gfCNCPoint5[22802] = {X 520.5269, Y 35.5815, Z -7.1667, A 0.000, B 0.000, C 0.000 }
gfCNCPoint5[22803] = {X 521.3531, Y 35.6727, Z -7.1667, A 0.000, B 0.000, C 0.000 }
gfCNCPoint5[22804] = {X 522.1466, Y 35.9205, Z -7.1667, A 0.000, B 0.000, C 0.000 }
gfCNCPoint5[22805] = {X 522.8780, Y 36.3157, Z -7.1667, A 0.000, B 0.000, C 0.000 }
gfCNCPoint5[22806] = {X 523.5201, Y 36.8436, Z -7.1667, A 0.000, B 0.000, C 0.000 }
gfCNCPoint5[22807] = {X 524.0492, Y 37.4848, Z -7.1667, A 0.000, B 0.000, C 0.000 }
gfCNCPoint5[22808] = {X 534.6319, Y 37.4851, Z -7.1667, A 0.000, B 0.000, C 0.000 }
gfCNCPoint5[22809] = {X 534.6319, Y 33.9662, Z -7.1667, A 0.000, B 0.000, C 0.000 }
gfCNCPoint5[22810] = {X 530.1083, Y 33.9675, Z -7.1667, A 0.000, B 0.000, C 0.000 }
gfCNCPoint5[22811] = {X 529.5761, Y 34.6112, Z -7.1667, A 0.000, B 0.000, C 0.000 }
gfCNCPoint5[22812] = {X 528.9300, Y 35.1404, Z -7.1667, A 0.000, B 0.000, C 0.000 }
gfCNCPoint5[22813] = {X 528.1941, Y 35.5354, Z -7.1667, A 0.000, B 0.000, C 0.000 }
gfCNCPoint5[22814] = {X 527.3960, Y 35.7814, Z -7.1667, A 0.000, B 0.000, C 0.000 }
gfCNCPoint5[22815] = {X 526.5655, Y 35.8693, Z -7.1667, A 0.000, B 0.000, C 0.000 }
gfCNCPoint5[22816] = {X 525.8868, Y 35.8694, Z -7.1667, A 0.000, B 0.000, C 0.000 }
gfCNCPoint5[22817] = {X 524.9255, Y 35.7611, Z -7.1667, A 0.000, B 0.000, C 0.000 }
gfCNCPoint5[22818] = {X 524.0124, Y 35.4416, Z -7.1667, A 0.000, B 0.000, C 0.000 }
gfCNCPoint5[22819] = {X 523.1933, Y 34.9270, Z -7.1667, A 0.000, B 0.000, C 0.000 }
gfCNCPoint5[22820] = {X 522.5092, Y 34.2429, Z -7.1667, A 0.000, B 0.000, C 0.000 }
gfCNCPoint5[22821] = {X 521.9946, Y 33.4238, Z -7.1667, A 0.000, B 0.000, C 0.000 }
gfCNCPoint5[22822] = {X 521.6751, Y 32.5107, Z -7.1667, A 0.000, B 0.000, C 0.000 }
gfCNCPoint5[22823] = {X 521.5668, Y 31.5495, Z -7.1667, A 0.000, B 0.000, C 0.000 }
gfCNCPoint5[22824] = {X 521.5668, Y 24.5714, Z -7.1667, A 0.000, B 0.000, C 0.000 }
gfCNCPoint5[22825] = {X 521.6739, Y 23.6153, Z -7.1667, A 0.000, B 0.000, C 0.000 }
gfCNCPoint5[22826] = {X 521.9900, Y 22.7066, Z -7.1667, A 0.000, B 0.000, C 0.000 }
gfCNCPoint5[22827] = {X 522.4994, Y 21.8904, Z -7.1667, A 0.000, B 0.000, C 0.000 }
gfCNCPoint5[22828] = {X 523.1768, Y 21.2071, Z -7.1667, A 0.000, B 0.000, C 0.000 }
gfCNCPoint5[22829] = {X 523.9886, Y 20.6908, Z -7.1667, A 0.000, B 0.000, C 0.000 }
gfCNCPoint5[22830] = {X 524.8946, Y 20.3669, Z -7.1667, A 0.000, B 0.000, C 0.000 }
gfCNCPoint5[22831] = {X 525.8498, Y 20.2516, Z -7.1667, A 0.000, B 0.000, C 0.000 }
gfCNCPoint5[22832] = {X 526.5695, Y 20.2516, Z -7.1667, A 0.000, B 0.000, C 0.000 }
gfCNCPoint5[22833] = {X 527.3943, Y 20.3391, Z -7.1667, A 0.000, B 0.000, C 0.000 }
gfCNCPoint5[22834] = {X 528.1872, Y 20.5826, Z -7.1667, A 0.000, B 0.000, C 0.000 }
gfCNCPoint5[22835] = {X 528.9190, Y 20.9731, Z -7.1667, A 0.000, B 0.000, C 0.000 }
gfCNCPoint5[22836] = {X 529.5626, Y 21.4964, Z -7.1667, A 0.000, B 0.000, C 0.000 }
gfCNCPoint5[22837] = {X 530.0944, Y 22.1329, Z -7.1667, A 0.000, B 0.000, C 0.000 }
gfCNCPoint5[22838] = {X 534.6319, Y 22.1331, Z -7.1667, A 0.000, B 0.000, C 0.000 }
gfCNCPoint5[22839] = {X 534.6319, Y 19.7026, Z -7.1667, A 0.000, B 0.000, C 0.000 }
gfCNCPoint5[22840] = {X 524.1915, Y 19.7025, Z -7.1667, A 0.000, B 0.000, C 0.000 }
gfCNCPoint5[22841] = {X 523.6591, Y 20.3468, Z -7.1667, A 0.000, B 0.000, C 0.000 }
gfCNCPoint5[22842] = {X 523.0125, Y 20.8765, Z -7.1667, A 0.000, B 0.000, C 0.000 }
gfCNCPoint5[22843] = {X 522.2760, Y 21.2718, Z -7.1667, A 0.000, B 0.000, C 0.000 }
gfCNCPoint5[22844] = {X 521.4772, Y 21.5179, Z -7.1667, A 0.000, B 0.000, C 0.000 }
gfCNCPoint5[22845] = {X 520.6460, Y 21.6056, Z -7.1667, A 0.000, B 0.000, C 0.000 }
gfCNCPoint5[22846] = {X 519.9691, Y 21.6057, Z -7.1667, A 0.000, B 0.000, C 0.000 }
gfCNCPoint5[22847] = {X 519.0078, Y 21.4974, Z -7.1667, A 0.000, B 0.000, C 0.000 }
gfCNCPoint5[22848] = {X 518.0947, Y 21.1779, Z -7.1667, A 0.000, B 0.000, C 0.000 }
gfCNCPoint5[22849] = {X 517.2756, Y 20.6632, Z -7.1667, A 0.000, B 0.000, C 0.000 }
gfCNCPoint5[22850] = {X 516.5916, Y 19.9792, Z -7.1667, A 0.000, B 0.000, C 0.000 }
gfCNCPoint5[22851] = {X 516.0769, Y 19.1601, Z -7.1667, A 0.000, B 0.000, C 0.000 }
gfCNCPoint5[22852] = {X 515.7574, Y 18.2470, Z -7.1667, A 0.000, B 0.000, C 0.000 }
gfCNCPoint5[22853] = {X 515.6491, Y 17.2857, Z -7.1667, A 0.000, B 0.000, C 0.000 }
gfCNCPoint5[22854] = {X 515.6491, Y 10.3077, Z -7.1667, A 0.000, B 0.000, C 0.000 }
gfCNCPoint5[22855] = {X 515.7562, Y 9.3519, Z -7.1667, A 0.000, B 0.000, C 0.000 }
gfCNCPoint5[22856] = {X 516.0720, Y 8.4435, Z -7.1667, A 0.000, B 0.000, C 0.000 }
gfCNCPoint5[22857] = {X 516.5811, Y 7.6275, Z -7.1667, A 0.000, B 0.000, C 0.000 }
gfCNCPoint5[22858] = {X 517.2580, Y 6.9443, Z -7.1667, A 0.000, B 0.000, C 0.000 }
gfCNCPoint5[22859] = {X 518.0693, Y 6.4278, Z -7.1667, A 0.000, B 0.000, C 0.000 }
gfCNCPoint5[22860] = {X 518.9748, Y 6.1037, Z -7.1667, A 0.000, B 0.000, C 0.000 }
gfCNCPoint5[22861] = {X 519.9296, Y 5.9879, Z -7.1667, A 0.000, B 0.000, C 0.000 }
gfCNCPoint5[22862] = {X 520.6502, Y 5.9879, Z -7.1667, A 0.000, B 0.000, C 0.000 }
gfCNCPoint5[22863] = {X 521.4754, Y 6.0751, Z -7.1667, A 0.000, B 0.000, C 0.000 }
gfCNCPoint5[22864] = {X 522.2687, Y 6.3185, Z -7.1667, A 0.000, B 0.000, C 0.000 }
gfCNCPoint5[22865] = {X 523.0008, Y 6.7091, Z -7.1667, A 0.000, B 0.000, C 0.000 }
gfCNCPoint5[22866] = {X 523.6448, Y 7.2324, Z -7.1667, A 0.000, B 0.000, C 0.000 }
gfCNCPoint5[22867] = {X 524.1768, Y 7.8692, Z -7.1667, A 0.000, B 0.000, C 0.000 }
gfCNCPoint5[22868] = {X 533.9633, Y 7.8694, Z -7.1667, A 0.000, B 0.000, C 0.000 }
gfCNCPoint5[22869] = {X 533.9634, Y 3.8694, Z -7.1667, A 0.000, B 0.000, C 0.000 }
gfCNCPoint5[22870] = {X 533.9633, Y 7.9494, Z -7.1667, A 0.000, B 0.000, C 0.000 }
gfCNCPoint5[22871] = {X 543.7510, Y 7.9496, Z -7.1667, A 0.000, B 0.000, C 0.000 }
gfCNCPoint5[22872] = {X 544.7134, Y 8.0333, Z -7.1667, A 0.000, B 0.000, C 0.000 }
gfCNCPoint5[22873] = {X 545.6320, Y 8.3325, Z -7.1667, A 0.000, B 0.000, C 0.000 }
gfCNCPoint5[22874] = {X 546.4591, Y 8.8316, Z -7.1667, A 0.000, B 0.000, C 0.000 }
gfCNCPoint5[22875] = {X 547.1520, Y 9.5048, Z -7.1667, A 0.000, B 0.000, C 0.000 }
gfCNCPoint5[22876] = {X 547.6747, Y 10.3173, Z -7.1667, A 0.000, B 0.000, C 0.000 }
gfCNCPoint5[22877] = {X 548.0001, Y 11.2269, Z -7.1667, A 0.000, B 0.000, C 0.000 }
gfCNCPoint5[22878] = {X 548.1114, Y 12.1865, Z -7.1667, A 0.000, B 0.000, C 0.000 }
gfCNCPoint5[22879] = {X 548.1112, Y 13.0217, Z -7.1667, A 0.000, B 0.000, C 0.000 }
gfCNCPoint5[22880] = {X 548.0029, Y 13.9312, Z -7.1667, A 0.000, B 0.000, C 0.000 }
gfCNCPoint5[22881] = {X 547.7018, Y 14.7962, Z -7.1667, A 0.000, B 0.000, C 0.000 }
gfCNCPoint5[22882] = {X 547.2220, Y 15.5764, Z -7.1667, A 0.000, B 0.000, C 0.000 }
gfCNCPoint5[22883] = {X 546.5858, Y 16.2353, Z -7.1667, A 0.000, B 0.000, C 0.000 }
gfCNCPoint5[22884] = {X 546.5850, Y 40.9520, Z -7.1667, A 0.000, B 0.000, C 0.000 }
gfCNCPoint5[22885] = {X 546.6353, Y 40.9934, Z -7.1667, A 0.000, B 0.000, C 0.000 }
gfCNCPoint5[22886] = {X 547.2529, Y 41.6508, Z -7.1667, A 0.000, B 0.000, C 0.000 }
gfCNCPoint5[22887] = {X 547.7175, Y 42.4239, Z -7.1667, A 0.000, B 0.000, C 0.000 }
gfCNCPoint5[22888] = {X 548.0080, Y 43.2779, Z -7.1667, A 0.000, B 0.000, C 0.000 }
gfCNCPoint5[22889] = {X 548.1113, Y 44.1740, Z -7.1667, A 0.000, B 0.000, C 0.000 }
gfCNCPoint5[22890] = {X 548.1114, Y 45.0003, Z -7.1667, A 0.000, B 0.000, C 0.000 }
gfCNCPoint5[22891] = {X 548.0001, Y 45.9599, Z -7.1667, A 0.000, B 0.000, C 0.000 }
gfCNCPoint5[22892] = {X 547.6746, Y 46.8695, Z -7.1667, A 0.000, B 0.000, C 0.000 }
gfCNCPoint5[22893] = {X 547.1519, Y 47.6819, Z -7.1667, A 0.000, B 0.000, C 0.000 }
gfCNCPoint5[22894] = {X 546.4591, Y 48.3551, Z -7.1667, A 0.000, B 0.000, C 0.000 }
gfCNCPoint5[22895] = {X 545.6320, Y 48.8541, Z -7.1667, A 0.000, B 0.000, C 0.000 }
gfCNCPoint5[22896] = {X 544.7134, Y 49.1533, Z -7.1667, A 0.000, B 0.000, C 0.000 }
gfCNCPoint5[22897] = {X 543.7510, Y 49.2369, Z -7.1667, A 0.000, B 0.000, C 0.000 }
gfCNCPoint5[22898] = {X 524.0041, Y 49.2373, Z -7.1667, A 0.000, B 0.000, C 0.000 }
gfCNCPoint5[22899] = {X 523.4672, Y 49.8705, Z -7.1667, A 0.000, B 0.000, C 0.000 }
gfCNCPoint5[22900] = {X 522.8209, Y 50.3914, Z -7.1667, A 0.000, B 0.000, C 0.000 }
gfCNCPoint5[22901] = {X 522.0882, Y 50.7816, Z -7.1667, A 0.000, B 0.000, C 0.000 }
gfCNCPoint5[22902] = {X 521.2952, Y 51.0271, Z -7.1667, A 0.000, B 0.000, C 0.000 }
gfCNCPoint5[22903] = {X 520.4702, Y 51.1191, Z -7.1667, A 0.000, B 0.000, C 0.000 }
gfCNCPoint5[22904] = {X 519.7998, Y 51.1191, Z -7.1667, A 0.000, B 0.000, C 0.000 }
gfCNCPoint5[22905] = {X 518.8563, Y 51.0128, Z -7.1667, A 0.000, B 0.000, C 0.000 }
gfCNCPoint5[22906] = {X 517.9601, Y 50.6992, Z -7.1667, A 0.000, B 0.000, C 0.000 }
gfCNCPoint5[22907] = {X 517.1562, Y 50.1941, Z -7.1667, A 0.000, B 0.000, C 0.000 }
gfCNCPoint5[22908] = {X 516.4848, Y 49.5227, Z -7.1667, A 0.000, B 0.000, C 0.000 }
gfCNCPoint5[22909] = {X 515.9797, Y 48.7188, Z -7.1667, A 0.000, B 0.000, C 0.000 }
gfCNCPoint5[22910] = {X 515.6661, Y 47.8226, Z -7.1667, A 0.000, B 0.000, C 0.000 }
gfCNCPoint5[22911] = {X 515.5598, Y 46.8791, Z -7.1667, A 0.000, B 0.000, C 0.000 }
gfCNCPoint5[22912] = {X 515.5598, Y 39.9011, Z -7.1667, A 0.000, B 0.000, C 0.000 }
gfCNCPoint5[22913] = {X 515.6649, Y 38.9628, Z -7.1667, A 0.000, B 0.000, C 0.000 }
gfCNCPoint5[22914] = {X 515.9751, Y 38.0710, Z -7.1667, A 0.000, B 0.000, C 0.000 }
gfCNCPoint5[22915] = {X 516.4749, Y 37.2700, Z -7.1667, A 0.000, B 0.000, C 0.000 }
gfCNCPoint5[22916] = {X 517.1395, Y 36.5995, Z -7.1667, A 0.000, B 0.000, C 0.000 }
gfCNCPoint5[22917] = {X 517.9361, Y 36.0926, Z -7.1667, A 0.000, B 0.000, C 0.000 }
gfCNCPoint5[22918] = {X 518.8251, Y 35.7746, Z -7.1667, A 0.000, B 0.000, C 0.000 }
gfCNCPoint5[22919] = {X 519.7624, Y 35.6613, Z -7.1667, A 0.000, B 0.000, C 0.000 }
gfCNCPoint5[22920] = {X 520.5258, Y 35.6615, Z -7.1667, A 0.000, B 0.000, C 0.000 }
gfCNCPoint5[22921] = {X 521.3450, Y 35.7528, Z -7.1667, A 0.000, B 0.000, C 0.000 }
gfCNCPoint5[22922] = {X 522.1312, Y 36.0008, Z -7.1667, A 0.000, B 0.000, C 0.000 }
gfCNCPoint5[22923] = {X 522.8544, Y 36.3963, Z -7.1667, A 0.000, B 0.000, C 0.000 }
gfCNCPoint5[22924] = {X 523.4875, Y 36.9243, Z -7.1667, A 0.000, B 0.000, C 0.000 }
gfCNCPoint5[22925] = {X 524.0064, Y 37.5648, Z -7.1667, A 0.000, B 0.000, C 0.000 }
gfCNCPoint5[22926] = {X 534.7119, Y 37.5651, Z -7.1667, A 0.000, B 0.000, C 0.000 }
gfCNCPoint5[22927] = {X 534.7119, Y 33.8862, Z -7.1667, A 0.000, B 0.000, C 0.000 }
gfCNCPoint5[22928] = {X 530.0654, Y 33.8860, Z -7.1667, A 0.000, B 0.000, C 0.000 }
gfCNCPoint5[22929] = {X 530.0414, Y 33.9236, Z -7.1667, A 0.000, B 0.000, C 0.000 }
gfCNCPoint5[22930] = {X 529.5191, Y 34.5550, Z -7.1667, A 0.000, B 0.000, C 0.000 }
gfCNCPoint5[22931] = {X 528.8850, Y 35.0742, Z -7.1667, A 0.000, B 0.000, C 0.000 }
gfCNCPoint5[22932] = {X 528.1629, Y 35.4617, Z -7.1667, A 0.000, B 0.000, C 0.000 }
gfCNCPoint5[22933] = {X 527.3797, Y 35.7031, Z -7.1667, A 0.000, B 0.000, C 0.000 }
gfCNCPoint5[22934] = {X 526.5648, Y 35.7893, Z -7.1667, A 0.000, B 0.000, C 0.000 }
gfCNCPoint5[22935] = {X 525.8868, Y 35.7894, Z -7.1667, A 0.000, B 0.000, C 0.000 }
gfCNCPoint5[22936] = {X 524.9433, Y 35.6831, Z -7.1667, A 0.000, B 0.000, C 0.000 }
gfCNCPoint5[22937] = {X 524.0471, Y 35.3696, Z -7.1667, A 0.000, B 0.000, C 0.000 }
gfCNCPoint5[22938] = {X 523.2432, Y 34.8644, Z -7.1667, A 0.000, B 0.000, C 0.000 }
gfCNCPoint5[22939] = {X 522.5718, Y 34.1930, Z -7.1667, A 0.000, B 0.000, C 0.000 }
gfCNCPoint5[22940] = {X 522.0666, Y 33.3891, Z -7.1667, A 0.000, B 0.000, C 0.000 }
gfCNCPoint5[22941] = {X 521.7531, Y 32.4929, Z -7.1667, A 0.000, B 0.000, C 0.000 }
gfCNCPoint5[22942] = {X 521.6468, Y 31.5495, Z -7.1667, A 0.000, B 0.000, C 0.000 }
gfCNCPoint5[22943] = {X 521.6468, Y 24.5714, Z -7.1667, A 0.000, B 0.000, C 0.000 }
gfCNCPoint5[22944] = {X 521.7519, Y 23.6330, Z -7.1667, A 0.000, B 0.000, C 0.000 }
gfCNCPoint5[22945] = {X 522.0622, Y 22.7411, Z -7.1667, A 0.000, B 0.000, C 0.000 }
gfCNCPoint5[22946] = {X 522.5621, Y 21.9400, Z -7.1667, A 0.000, B 0.000, C 0.000 }
gfCNCPoint5[22947] = {X 523.2270, Y 21.2694, Z -7.1667, A 0.000, B 0.000, C 0.000 }
gfCNCPoint5[22948] = {X 524.0238, Y 20.7626, Z -7.1667, A 0.000, B 0.000, C 0.000 }
gfCNCPoint5[22949] = {X 524.9130, Y 20.4448, Z -7.1667, A 0.000, B 0.000, C 0.000 }
gfCNCPoint5[22950] = {X 525.8505, Y 20.3316, Z -7.1667, A 0.000, B 0.000, C 0.000 }
gfCNCPoint5[22951] = {X 526.5687, Y 20.3316, Z -7.1667, A 0.000, B 0.000, C 0.000 }
gfCNCPoint5[22952] = {X 527.3865, Y 20.4192, Z -7.1667, A 0.000, B 0.000, C 0.000 }
gfCNCPoint5[22953] = {X 528.1720, Y 20.6630, Z -7.1667, A 0.000, B 0.000, C 0.000 }
gfCNCPoint5[22954] = {X 528.8957, Y 21.0538, Z -7.1667, A 0.000, B 0.000, C 0.000 }
gfCNCPoint5[22955] = {X 529.5303, Y 21.5770, Z -7.1667, A 0.000, B 0.000, C 0.000 }
gfCNCPoint5[22956] = {X 530.0519, Y 22.2129, Z -7.1667, A 0.000, B 0.000, C 0.000 }
gfCNCPoint5[22957] = {X 534.7119, Y 22.2131, Z -7.1667, A 0.000, B 0.000, C 0.000 }
gfCNCPoint5[22958] = {X 534.7119, Y 19.6226, Z -7.1667, A 0.000, B 0.000, C 0.000 }
gfCNCPoint5[22959] = {X 524.1486, Y 19.6225, Z -7.1667, A 0.000, B 0.000, C 0.000 }
gfCNCPoint5[22960] = {X 524.1252, Y 19.6577, Z -7.1667, A 0.000, B 0.000, C 0.000 }
gfCNCPoint5[22961] = {X 523.6026, Y 20.2901, Z -7.1667, A 0.000, B 0.000, C 0.000 }
gfCNCPoint5[22962] = {X 522.9680, Y 20.8100, Z -7.1667, A 0.000, B 0.000, C 0.000 }
gfCNCPoint5[22963] = {X 522.2452, Y 21.1980, Z -7.1667, A 0.000, B 0.000, C 0.000 }
gfCNCPoint5[22964] = {X 521.4612, Y 21.4396, Z -7.1667, A 0.000, B 0.000, C 0.000 }
gfCNCPoint5[22965] = {X 520.6453, Y 21.5256, Z -7.1667, A 0.000, B 0.000, C 0.000 }
gfCNCPoint5[22966] = {X 519.9691, Y 21.5257, Z -7.1667, A 0.000, B 0.000, C 0.000 }
gfCNCPoint5[22967] = {X 519.0256, Y 21.4194, Z -7.1667, A 0.000, B 0.000, C 0.000 }
gfCNCPoint5[22968] = {X 518.1294, Y 21.1058, Z -7.1667, A 0.000, B 0.000, C 0.000 }
gfCNCPoint5[22969] = {X 517.3255, Y 20.6007, Z -7.1667, A 0.000, B 0.000, C 0.000 }
gfCNCPoint5[22970] = {X 516.6541, Y 19.9293, Z -7.1667, A 0.000, B 0.000, C 0.000 }
gfCNCPoint5[22971] = {X 516.1490, Y 19.1254, Z -7.1667, A 0.000, B 0.000, C 0.000 }
gfCNCPoint5[22972] = {X 515.8354, Y 18.2292, Z -7.1667, A 0.000, B 0.000, C 0.000 }
gfCNCPoint5[22973] = {X 515.7291, Y 17.2857, Z -7.1667, A 0.000, B 0.000, C 0.000 }
gfCNCPoint5[22974] = {X 515.7291, Y 10.3077, Z -7.1667, A 0.000, B 0.000, C 0.000 }
gfCNCPoint5[22975] = {X 515.8342, Y 9.3696, Z -7.1667, A 0.000, B 0.000, C 0.000 }
gfCNCPoint5[22976] = {X 516.1442, Y 8.4780, Z -7.1667, A 0.000, B 0.000, C 0.000 }
gfCNCPoint5[22977] = {X 516.6438, Y 7.6771, Z -7.1667, A 0.000, B 0.000, C 0.000 }
gfCNCPoint5[22978] = {X 517.3082, Y 7.0066, Z -7.1667, A 0.000, B 0.000, C 0.000 }
gfCNCPoint5[22979] = {X 518.1045, Y 6.4997, Z -7.1667, A 0.000, B 0.000, C 0.000 }
gfCNCPoint5[22980] = {X 518.9932, Y 6.1815, Z -7.1667, A 0.000, B 0.000, C 0.000 }
gfCNCPoint5[22981] = {X 519.9303, Y 6.0679, Z -7.1667, A 0.000, B 0.000, C 0.000 }
gfCNCPoint5[22982] = {X 520.6494, Y 6.0679, Z -7.1667, A 0.000, B 0.000, C 0.000 }
gfCNCPoint5[22983] = {X 521.4676, Y 6.1552, Z -7.1667, A 0.000, B 0.000, C 0.000 }
gfCNCPoint5[22984] = {X 522.2535, Y 6.3988, Z -7.1667, A 0.000, B 0.000, C 0.000 }
gfCNCPoint5[22985] = {X 522.9775, Y 6.7897, Z -7.1667, A 0.000, B 0.000, C 0.000 }
gfCNCPoint5[22986] = {X 523.6124, Y 7.3131, Z -7.1667, A 0.000, B 0.000, C 0.000 }
gfCNCPoint5[22987] = {X 524.1343, Y 7.9492, Z -7.1667, A 0.000, B 0.000, C 0.000 }
gfCNCPoint5[22988] = {X 533.9633, Y 7.9494, Z -7.1667, A 0.000, B 0.000, C 0.000 }
gfCNCPoint5[22989] = {X 533.9634, Y 3.9494, Z -7.1667, A 0.000, B 0.000, C 0.000 }
gfCNCPoint5[22990] = {X 533.9633, Y 8.0294, Z -7.1667, A 0.000, B 0.000, C 0.000 }
gfCNCPoint5[22991] = {X 543.7521, Y 8.0296, Z -7.1667, A 0.000, B 0.000, C 0.000 }
gfCNCPoint5[22992] = {X 544.6966, Y 8.1115, Z -7.1667, A 0.000, B 0.000, C 0.000 }
gfCNCPoint5[22993] = {X 545.5980, Y 8.4049, Z -7.1667, A 0.000, B 0.000, C 0.000 }
gfCNCPoint5[22994] = {X 546.4098, Y 8.8946, Z -7.1667, A 0.000, B 0.000, C 0.000 }
gfCNCPoint5[22995] = {X 547.0898, Y 9.5551, Z -7.1667, A 0.000, B 0.000, C 0.000 }
gfCNCPoint5[22996] = {X 547.6028, Y 10.3523, Z -7.1667, A 0.000, B 0.000, C 0.000 }
gfCNCPoint5[22997] = {X 547.9222, Y 11.2449, Z -7.1667, A 0.000, B 0.000, C 0.000 }
gfCNCPoint5[22998] = {X 548.0314, Y 12.1866, Z -7.1667, A 0.000, B 0.000, C 0.000 }
gfCNCPoint5[22999] = {X 548.0312, Y 13.0208, Z -7.1667, A 0.000, B 0.000, C 0.000 }
gfCNCPoint5[23000] = {X 547.9228, Y 13.9223, Z -7.1667, A 0.000, B 0.000, C 0.000 }
gfCNCPoint5[23001] = {X 547.6215, Y 14.7787, Z -7.1667, A 0.000, B 0.000, C 0.000 }
gfCNCPoint5[23002] = {X 547.1415, Y 15.5494, Z -7.1667, A 0.000, B 0.000, C 0.000 }
gfCNCPoint5[23003] = {X 546.5058, Y 16.1976, Z -7.1667, A 0.000, B 0.000, C 0.000 }
gfCNCPoint5[23004] = {X 546.5050, Y 40.9898, Z -7.1667, A 0.000, B 0.000, C 0.000 }
gfCNCPoint5[23005] = {X 546.5838, Y 41.0546, Z -7.1667, A 0.000, B 0.000, C 0.000 }
gfCNCPoint5[23006] = {X 547.1895, Y 41.6996, Z -7.1667, A 0.000, B 0.000, C 0.000 }
gfCNCPoint5[23007] = {X 547.6451, Y 42.4580, Z -7.1667, A 0.000, B 0.000, C 0.000 }
gfCNCPoint5[23008] = {X 547.9300, Y 43.2957, Z -7.1667, A 0.000, B 0.000, C 0.000 }
gfCNCPoint5[23009] = {X 548.0313, Y 44.1746, Z -7.1667, A 0.000, B 0.000, C 0.000 }
gfCNCPoint5[23010] = {X 548.0314, Y 45.0002, Z -7.1667, A 0.000, B 0.000, C 0.000 }
gfCNCPoint5[23011] = {X 547.9221, Y 45.9419, Z -7.1667, A 0.000, B 0.000, C 0.000 }
gfCNCPoint5[23012] = {X 547.6027, Y 46.8344, Z -7.1667, A 0.000, B 0.000, C 0.000 }
gfCNCPoint5[23013] = {X 547.0897, Y 47.6316, Z -7.1667, A 0.000, B 0.000, C 0.000 }
gfCNCPoint5[23014] = {X 546.4097, Y 48.2921, Z -7.1667, A 0.000, B 0.000, C 0.000 }
gfCNCPoint5[23015] = {X 545.5980, Y 48.7817, Z -7.1667, A 0.000, B 0.000, C 0.000 }
gfCNCPoint5[23016] = {X 544.6965, Y 49.0750, Z -7.1667, A 0.000, B 0.000, C 0.000 }
gfCNCPoint5[23017] = {X 543.7521, Y 49.1569, Z -7.1667, A 0.000, B 0.000, C 0.000 }
gfCNCPoint5[23018] = {X 523.9621, Y 49.1573, Z -7.1667, A 0.000, B 0.000, C 0.000 }
gfCNCPoint5[23019] = {X 523.4352, Y 49.7898, Z -7.1667, A 0.000, B 0.000, C 0.000 }
gfCNCPoint5[23020] = {X 522.7978, Y 50.3107, Z -7.1667, A 0.000, B 0.000, C 0.000 }
gfCNCPoint5[23021] = {X 522.0731, Y 50.7012, Z -7.1667, A 0.000, B 0.000, C 0.000 }
gfCNCPoint5[23022] = {X 521.2875, Y 50.9470, Z -7.1667, A 0.000, B 0.000, C 0.000 }
gfCNCPoint5[23023] = {X 520.4695, Y 51.0391, Z -7.1667, A 0.000, B 0.000, C 0.000 }
gfCNCPoint5[23024] = {X 519.7998, Y 51.0391, Z -7.1667, A 0.000, B 0.000, C 0.000 }
gfCNCPoint5[23025] = {X 518.8741, Y 50.9348, Z -7.1667, A 0.000, B 0.000, C 0.000 }
gfCNCPoint5[23026] = {X 517.9948, Y 50.6272, Z -7.1667, A 0.000, B 0.000, C 0.000 }
gfCNCPoint5[23027] = {X 517.2061, Y 50.1315, Z -7.1667, A 0.000, B 0.000, C 0.000 }
gfCNCPoint5[23028] = {X 516.5474, Y 49.4728, Z -7.1667, A 0.000, B 0.000, C 0.000 }
gfCNCPoint5[23029] = {X 516.0517, Y 48.6841, Z -7.1667, A 0.000, B 0.000, C 0.000 }
gfCNCPoint5[23030] = {X 515.7441, Y 47.8048, Z -7.1667, A 0.000, B 0.000, C 0.000 }
gfCNCPoint5[23031] = {X 515.6398, Y 46.8791, Z -7.1667, A 0.000, B 0.000, C 0.000 }
gfCNCPoint5[23032] = {X 515.6398, Y 39.9011, Z -7.1667, A 0.000, B 0.000, C 0.000 }
gfCNCPoint5[23033] = {X 515.7429, Y 38.9805, Z -7.1667, A 0.000, B 0.000, C 0.000 }
gfCNCPoint5[23034] = {X 516.0472, Y 38.1056, Z -7.1667, A 0.000, B 0.000, C 0.000 }
gfCNCPoint5[23035] = {X 516.5376, Y 37.3197, Z -7.1667, A 0.000, B 0.000, C 0.000 }
gfCNCPoint5[23036] = {X 517.1897, Y 36.6618, Z -7.1667, A 0.000, B 0.000, C 0.000 }
gfCNCPoint5[23037] = {X 517.9713, Y 36.1645, Z -7.1667, A 0.000, B 0.000, C 0.000 }
gfCNCPoint5[23038] = {X 518.8435, Y 35.8525, Z -7.1667, A 0.000, B 0.000, C 0.000 }
gfCNCPoint5[23039] = {X 519.7631, Y 35.7413, Z -7.1667, A 0.000, B 0.000, C 0.000 }
gfCNCPoint5[23040] = {X 520.5247, Y 35.7415, Z -7.1667, A 0.000, B 0.000, C 0.000 }
gfCNCPoint5[23041] = {X 521.3369, Y 35.8328, Z -7.1667, A 0.000, B 0.000, C 0.000 }
gfCNCPoint5[23042] = {X 522.1156, Y 36.0812, Z -7.1667, A 0.000, B 0.000, C 0.000 }
gfCNCPoint5[23043] = {X 522.8306, Y 36.4770, Z -7.1667, A 0.000, B 0.000, C 0.000 }
gfCNCPoint5[23044] = {X 523.4545, Y 37.0050, Z -7.1667, A 0.000, B 0.000, C 0.000 }
gfCNCPoint5[23045] = {X 523.9631, Y 37.6448, Z -7.1667, A 0.000, B 0.000, C 0.000 }
gfCNCPoint5[23046] = {X 534.7919, Y 37.6451, Z -7.1667, A 0.000, B 0.000, C 0.000 }
gfCNCPoint5[23047] = {X 534.7919, Y 33.8062, Z -7.1667, A 0.000, B 0.000, C 0.000 }
gfCNCPoint5[23048] = {X 530.0216, Y 33.8060, Z -7.1667, A 0.000, B 0.000, C 0.000 }
gfCNCPoint5[23049] = {X 529.9746, Y 33.8796, Z -7.1667, A 0.000, B 0.000, C 0.000 }
gfCNCPoint5[23050] = {X 529.4621, Y 34.4989, Z -7.1667, A 0.000, B 0.000, C 0.000 }
gfCNCPoint5[23051] = {X 528.8400, Y 35.0081, Z -7.1667, A 0.000, B 0.000, C 0.000 }
gfCNCPoint5[23052] = {X 528.1317, Y 35.3881, Z -7.1667, A 0.000, B 0.000, C 0.000 }
gfCNCPoint5[23053] = {X 527.3635, Y 35.6248, Z -7.1667, A 0.000, B 0.000, C 0.000 }
gfCNCPoint5[23054] = {X 526.5641, Y 35.7093, Z -7.1667, A 0.000, B 0.000, C 0.000 }
gfCNCPoint5[23055] = {X 525.8868, Y 35.7095, Z -7.1667, A 0.000, B 0.000, C 0.000 }
gfCNCPoint5[23056] = {X 524.9611, Y 35.6052, Z -7.1667, A 0.000, B 0.000, C 0.000 }
gfCNCPoint5[23057] = {X 524.0818, Y 35.2975, Z -7.1667, A 0.000, B 0.000, C 0.000 }
gfCNCPoint5[23058] = {X 523.2930, Y 34.8019, Z -7.1667, A 0.000, B 0.000, C 0.000 }
gfCNCPoint5[23059] = {X 522.6343, Y 34.1432, Z -7.1667, A 0.000, B 0.000, C 0.000 }
gfCNCPoint5[23060] = {X 522.1387, Y 33.3544, Z -7.1667, A 0.000, B 0.000, C 0.000 }
gfCNCPoint5[23061] = {X 521.8311, Y 32.4751, Z -7.1667, A 0.000, B 0.000, C 0.000 }
gfCNCPoint5[23062] = {X 521.7268, Y 31.5495, Z -7.1667, A 0.000, B 0.000, C 0.000 }
gfCNCPoint5[23063] = {X 521.7268, Y 24.5714, Z -7.1667, A 0.000, B 0.000, C 0.000 }
gfCNCPoint5[23064] = {X 521.8299, Y 23.6507, Z -7.1667, A 0.000, B 0.000, C 0.000 }
gfCNCPoint5[23065] = {X 522.1343, Y 22.7756, Z -7.1667, A 0.000, B 0.000, C 0.000 }
gfCNCPoint5[23066] = {X 522.6248, Y 21.9897, Z -7.1667, A 0.000, B 0.000, C 0.000 }
gfCNCPoint5[23067] = {X 523.2772, Y 21.3317, Z -7.1667, A 0.000, B 0.000, C 0.000 }
gfCNCPoint5[23068] = {X 524.0589, Y 20.8345, Z -7.1667, A 0.000, B 0.000, C 0.000 }
gfCNCPoint5[23069] = {X 524.9313, Y 20.5226, Z -7.1667, A 0.000, B 0.000, C 0.000 }
gfCNCPoint5[23070] = {X 525.8511, Y 20.4116, Z -7.1667, A 0.000, B 0.000, C 0.000 }
gfCNCPoint5[23071] = {X 526.5679, Y 20.4116, Z -7.1667, A 0.000, B 0.000, C 0.000 }
gfCNCPoint5[23072] = {X 527.3787, Y 20.4992, Z -7.1667, A 0.000, B 0.000, C 0.000 }
gfCNCPoint5[23073] = {X 528.1567, Y 20.7433, Z -7.1667, A 0.000, B 0.000, C 0.000 }
gfCNCPoint5[23074] = {X 528.8722, Y 21.1345, Z -7.1667, A 0.000, B 0.000, C 0.000 }
gfCNCPoint5[23075] = {X 529.4976, Y 21.6577, Z -7.1667, A 0.000, B 0.000, C 0.000 }
gfCNCPoint5[23076] = {X 530.0089, Y 22.2929, Z -7.1667, A 0.000, B 0.000, C 0.000 }
gfCNCPoint5[23077] = {X 534.7919, Y 22.2931, Z -7.1667, A 0.000, B 0.000, C 0.000 }
gfCNCPoint5[23078] = {X 534.7919, Y 19.5426, Z -7.1667, A 0.000, B 0.000, C 0.000 }
gfCNCPoint5[23079] = {X 524.1048, Y 19.5425, Z -7.1667, A 0.000, B 0.000, C 0.000 }
gfCNCPoint5[23080] = {X 524.0760, Y 19.5874, Z -7.1667, A 0.000, B 0.000, C 0.000 }
gfCNCPoint5[23081] = {X 523.5636, Y 20.2160, Z -7.1667, A 0.000, B 0.000, C 0.000 }
gfCNCPoint5[23082] = {X 522.9389, Y 20.7332, Z -7.1667, A 0.000, B 0.000, C 0.000 }
gfCNCPoint5[23083] = {X 522.2257, Y 21.1194, Z -7.1667, A 0.000, B 0.000, C 0.000 }
gfCNCPoint5[23084] = {X 521.4512, Y 21.3599, Z -7.1667, A 0.000, B 0.000, C 0.000 }
gfCNCPoint5[23085] = {X 520.6447, Y 21.4456, Z -7.1667, A 0.000, B 0.000, C 0.000 }
gfCNCPoint5[23086] = {X 519.9691, Y 21.4457, Z -7.1667, A 0.000, B 0.000, C 0.000 }
gfCNCPoint5[23087] = {X 519.0434, Y 21.3414, Z -7.1667, A 0.000, B 0.000, C 0.000 }
gfCNCPoint5[23088] = {X 518.1641, Y 21.0337, Z -7.1667, A 0.000, B 0.000, C 0.000 }
gfCNCPoint5[23089] = {X 517.3754, Y 20.5381, Z -7.1667, A 0.000, B 0.000, C 0.000 }
gfCNCPoint5[23090] = {X 516.7167, Y 19.8794, Z -7.1667, A 0.000, B 0.000, C 0.000 }
gfCNCPoint5[23091] = {X 516.2211, Y 19.0907, Z -7.1667, A 0.000, B 0.000, C 0.000 }
gfCNCPoint5[23092] = {X 515.9134, Y 18.2114, Z -7.1667, A 0.000, B 0.000, C 0.000 }
gfCNCPoint5[23093] = {X 515.8091, Y 17.2857, Z -7.1667, A 0.000, B 0.000, C 0.000 }
gfCNCPoint5[23094] = {X 515.8091, Y 10.3077, Z -7.1667, A 0.000, B 0.000, C 0.000 }
gfCNCPoint5[23095] = {X 515.9122, Y 9.3873, Z -7.1667, A 0.000, B 0.000, C 0.000 }
gfCNCPoint5[23096] = {X 516.2164, Y 8.5125, Z -7.1667, A 0.000, B 0.000, C 0.000 }
gfCNCPoint5[23097] = {X 516.7065, Y 7.7267, Z -7.1667, A 0.000, B 0.000, C 0.000 }
gfCNCPoint5[23098] = {X 517.3584, Y 7.0689, Z -7.1667, A 0.000, B 0.000, C 0.000 }
gfCNCPoint5[23099] = {X 518.1397, Y 6.5715, Z -7.1667, A 0.000, B 0.000, C 0.000 }
gfCNCPoint5[23100] = {X 519.0117, Y 6.2594, Z -7.1667, A 0.000, B 0.000, C 0.000 }
gfCNCPoint5[23101] = {X 519.9311, Y 6.1479, Z -7.1667, A 0.000, B 0.000, C 0.000 }
gfCNCPoint5[23102] = {X 520.6487, Y 6.1479, Z -7.1667, A 0.000, B 0.000, C 0.000 }
gfCNCPoint5[23103] = {X 521.4598, Y 6.2352, Z -7.1667, A 0.000, B 0.000, C 0.000 }
gfCNCPoint5[23104] = {X 522.2382, Y 6.4792, Z -7.1667, A 0.000, B 0.000, C 0.000 }
gfCNCPoint5[23105] = {X 522.9540, Y 6.8704, Z -7.1667, A 0.000, B 0.000, C 0.000 }
gfCNCPoint5[23106] = {X 523.5798, Y 7.3938, Z -7.1667, A 0.000, B 0.000, C 0.000 }
gfCNCPoint5[23107] = {X 524.0913, Y 8.0292, Z -7.1667, A 0.000, B 0.000, C 0.000 }
gfCNCPoint5[23108] = {X 533.9633, Y 8.0294, Z -7.1667, A 0.000, B 0.000, C 0.000 }
gfCNCPoint5[23109] = {X 533.9634, Y 4.0294, Z -7.1667, A 0.000, B 0.000, C 0.000 }
gfCNCPoint5[23110] = {X 533.9633, Y 8.1094, Z -7.1667, A 0.000, B 0.000, C 0.000 }
gfCNCPoint5[23111] = {X 543.7532, Y 8.1096, Z -7.1667, A 0.000, B 0.000, C 0.000 }
gfCNCPoint5[23112] = {X 544.6797, Y 8.1897, Z -7.1667, A 0.000, B 0.000, C 0.000 }
gfCNCPoint5[23113] = {X 545.5641, Y 8.4773, Z -7.1667, A 0.000, B 0.000, C 0.000 }
gfCNCPoint5[23114] = {X 546.3604, Y 8.9575, Z -7.1667, A 0.000, B 0.000, C 0.000 }
gfCNCPoint5[23115] = {X 547.0276, Y 9.6054, Z -7.1667, A 0.000, B 0.000, C 0.000 }
gfCNCPoint5[23116] = {X 547.5308, Y 10.3874, Z -7.1667, A 0.000, B 0.000, C 0.000 }
gfCNCPoint5[23117] = {X 547.8442, Y 11.2630, Z -7.1667, A 0.000, B 0.000, C 0.000 }
gfCNCPoint5[23118] = {X 547.9514, Y 12.1867, Z -7.1667, A 0.000, B 0.000, C 0.000 }
gfCNCPoint5[23119] = {X 547.9512, Y 13.0200, Z -7.1667, A 0.000, B 0.000, C 0.000 }
gfCNCPoint5[23120] = {X 547.8428, Y 13.9133, Z -7.1667, A 0.000, B 0.000, C 0.000 }
gfCNCPoint5[23121] = {X 547.5412, Y 14.7611, Z -7.1667, A 0.000, B 0.000, C 0.000 }
gfCNCPoint5[23122] = {X 547.0611, Y 15.5222, Z -7.1667, A 0.000, B 0.000, C 0.000 }
gfCNCPoint5[23123] = {X 546.4258, Y 16.1595, Z -7.1667, A 0.000, B 0.000, C 0.000 }
gfCNCPoint5[23124] = {X 546.4250, Y 41.0276, Z -7.1667, A 0.000, B 0.000, C 0.000 }
gfCNCPoint5[23125] = {X 546.5323, Y 41.1158, Z -7.1667, A 0.000, B 0.000, C 0.000 }
gfCNCPoint5[23126] = {X 547.1260, Y 41.7483, Z -7.1667, A 0.000, B 0.000, C 0.000 }
gfCNCPoint5[23127] = {X 547.5727, Y 42.4921, Z -7.1667, A 0.000, B 0.000, C 0.000 }
gfCNCPoint5[23128] = {X 547.8520, Y 43.3134, Z -7.1667, A 0.000, B 0.000, C 0.000 }
gfCNCPoint5[23129] = {X 547.9513, Y 44.1753, Z -7.1667, A 0.000, B 0.000, C 0.000 }
gfCNCPoint5[23130] = {X 547.9514, Y 45.0001, Z -7.1667, A 0.000, B 0.000, C 0.000 }
gfCNCPoint5[23131] = {X 547.8442, Y 45.9238, Z -7.1667, A 0.000, B 0.000, C 0.000 }
gfCNCPoint5[23132] = {X 547.5308, Y 46.7993, Z -7.1667, A 0.000, B 0.000, C 0.000 }
gfCNCPoint5[23133] = {X 547.0275, Y 47.5813, Z -7.1667, A 0.000, B 0.000, C 0.000 }
gfCNCPoint5[23134] = {X 546.3604, Y 48.2291, Z -7.1667, A 0.000, B 0.000, C 0.000 }
gfCNCPoint5[23135] = {X 545.5640, Y 48.7093, Z -7.1667, A 0.000, B 0.000, C 0.000 }
gfCNCPoint5[23136] = {X 544.6797, Y 48.9968, Z -7.1667, A 0.000, B 0.000, C 0.000 }
gfCNCPoint5[23137] = {X 543.7532, Y 49.0769, Z -7.1667, A 0.000, B 0.000, C 0.000 }
gfCNCPoint5[23138] = {X 523.9196, Y 49.0773, Z -7.1667, A 0.000, B 0.000, C 0.000 }
gfCNCPoint5[23139] = {X 523.4028, Y 49.7090, Z -7.1667, A 0.000, B 0.000, C 0.000 }
gfCNCPoint5[23140] = {X 522.7745, Y 50.2300, Z -7.1667, A 0.000, B 0.000, C 0.000 }
gfCNCPoint5[23141] = {X 522.0580, Y 50.6207, Z -7.1667, A 0.000, B 0.000, C 0.000 }
gfCNCPoint5[23142] = {X 521.2798, Y 50.8668, Z -7.1667, A 0.000, B 0.000, C 0.000 }
gfCNCPoint5[23143] = {X 520.4688, Y 50.9591, Z -7.1667, A 0.000, B 0.000, C 0.000 }
gfCNCPoint5[23144] = {X 519.7998, Y 50.9591, Z -7.1667, A 0.000, B 0.000, C 0.000 }
gfCNCPoint5[23145] = {X 518.8919, Y 50.8568, Z -7.1667, A 0.000, B 0.000, C 0.000 }
gfCNCPoint5[23146] = {X 518.0295, Y 50.5551, Z -7.1667, A 0.000, B 0.000, C 0.000 }
gfCNCPoint5[23147] = {X 517.2559, Y 50.0690, Z -7.1667, A 0.000, B 0.000, C 0.000 }
gfCNCPoint5[23148] = {X 516.6099, Y 49.4230, Z -7.1667, A 0.000, B 0.000, C 0.000 }
gfCNCPoint5[23149] = {X 516.1238, Y 48.6494, Z -7.1667, A 0.000, B 0.000, C 0.000 }
gfCNCPoint5[23150] = {X 515.8221, Y 47.7870, Z -7.1667, A 0.000, B 0.000, C 0.000 }
gfCNCPoint5[23151] = {X 515.7198, Y 46.8791, Z -7.1667, A 0.000, B 0.000, C 0.000 }
gfCNCPoint5[23152] = {X 515.7198, Y 39.9011, Z -7.1667, A 0.000, B 0.000, C 0.000 }
gfCNCPoint5[23153] = {X 515.8209, Y 38.9982, Z -7.1667, A 0.000, B 0.000, C 0.000 }
gfCNCPoint5[23154] = {X 516.1194, Y 38.1401, Z -7.1667, A 0.000, B 0.000, C 0.000 }
gfCNCPoint5[23155] = {X 516.6003, Y 37.3693, Z -7.1667, A 0.000, B 0.000, C 0.000 }
gfCNCPoint5[23156] = {X 517.2399, Y 36.7241, Z -7.1667, A 0.000, B 0.000, C 0.000 }
gfCNCPoint5[23157] = {X 518.0064, Y 36.2364, Z -7.1667, A 0.000, B 0.000, C 0.000 }
gfCNCPoint5[23158] = {X 518.8619, Y 35.9304, Z -7.1667, A 0.000, B 0.000, C 0.000 }
gfCNCPoint5[23159] = {X 519.7638, Y 35.8213, Z -7.1667, A 0.000, B 0.000, C 0.000 }
gfCNCPoint5[23160] = {X 520.5236, Y 35.8215, Z -7.1667, A 0.000, B 0.000, C 0.000 }
gfCNCPoint5[23161] = {X 521.3287, Y 35.9129, Z -7.1667, A 0.000, B 0.000, C 0.000 }
gfCNCPoint5[23162] = {X 522.0998, Y 36.1616, Z -7.1667, A 0.000, B 0.000, C 0.000 }
gfCNCPoint5[23163] = {X 522.8066, Y 36.5577, Z -7.1667, A 0.000, B 0.000, C 0.000 }
gfCNCPoint5[23164] = {X 523.4212, Y 37.0857, Z -7.1667, A 0.000, B 0.000, C 0.000 }
gfCNCPoint5[23165] = {X 523.9193, Y 37.7248, Z -7.1667, A 0.000, B 0.000, C 0.000 }
gfCNCPoint5[23166] = {X 534.8719, Y 37.7251, Z -7.1667, A 0.000, B 0.000, C 0.000 }
gfCNCPoint5[23167] = {X 534.8719, Y 33.7262, Z -7.1667, A 0.000, B 0.000, C 0.000 }
gfCNCPoint5[23168] = {X 529.9777, Y 33.7260, Z -7.1667, A 0.000, B 0.000, C 0.000 }
gfCNCPoint5[23169] = {X 529.9071, Y 33.8366, Z -7.1667, A 0.000, B 0.000, C 0.000 }
gfCNCPoint5[23170] = {X 529.2612, Y 34.5790, Z -7.1667, A 0.000, B 0.000, C 0.000 }
gfCNCPoint5[23171] = {X 528.4563, Y 35.1452, Z -7.1667, A 0.000, B 0.000, C 0.000 }
gfCNCPoint5[23172] = {X 527.5392, Y 35.5023, Z -7.1667, A 0.000, B 0.000, C 0.000 }
gfCNCPoint5[23173] = {X 526.5634, Y 35.6293, Z -7.1667, A 0.000, B 0.000, C 0.000 }
gfCNCPoint5[23174] = {X 525.8868, Y 35.6295, Z -7.1667, A 0.000, B 0.000, C 0.000 }
gfCNCPoint5[23175] = {X 524.9789, Y 35.5272, Z -7.1667, A 0.000, B 0.000, C 0.000 }
gfCNCPoint5[23176] = {X 524.1165, Y 35.2254, Z -7.1667, A 0.000, B 0.000, C 0.000 }
gfCNCPoint5[23177] = {X 523.3429, Y 34.7393, Z -7.1667, A 0.000, B 0.000, C 0.000 }
gfCNCPoint5[23178] = {X 522.6969, Y 34.0933, Z -7.1667, A 0.000, B 0.000, C 0.000 }
gfCNCPoint5[23179] = {X 522.2108, Y 33.3197, Z -7.1667, A 0.000, B 0.000, C 0.000 }
gfCNCPoint5[23180] = {X 521.9091, Y 32.4573, Z -7.1667, A 0.000, B 0.000, C 0.000 }
gfCNCPoint5[23181] = {X 521.8068, Y 31.5495, Z -7.1667, A 0.000, B 0.000, C 0.000 }
gfCNCPoint5[23182] = {X 521.8068, Y 24.5714, Z -7.1667, A 0.000, B 0.000, C 0.000 }
gfCNCPoint5[23183] = {X 521.9079, Y 23.6684, Z -7.1667, A 0.000, B 0.000, C 0.000 }
gfCNCPoint5[23184] = {X 522.2065, Y 22.8102, Z -7.1667, A 0.000, B 0.000, C 0.000 }
gfCNCPoint5[23185] = {X 522.6876, Y 22.0393, Z -7.1667, A 0.000, B 0.000, C 0.000 }
gfCNCPoint5[23186] = {X 523.3273, Y 21.3940, Z -7.1667, A 0.000, B 0.000, C 0.000 }
gfCNCPoint5[23187] = {X 524.0941, Y 20.9064, Z -7.1667, A 0.000, B 0.000, C 0.000 }
gfCNCPoint5[23188] = {X 524.9497, Y 20.6005, Z -7.1667, A 0.000, B 0.000, C 0.000 }
gfCNCPoint5[23189] = {X 525.8518, Y 20.4916, Z -7.1667, A 0.000, B 0.000, C 0.000 }
gfCNCPoint5[23190] = {X 526.5672, Y 20.4916, Z -7.1667, A 0.000, B 0.000, C 0.000 }
gfCNCPoint5[23191] = {X 527.3707, Y 20.5793, Z -7.1667, A 0.000, B 0.000, C 0.000 }
gfCNCPoint5[23192] = {X 528.1412, Y 20.8237, Z -7.1667, A 0.000, B 0.000, C 0.000 }
gfCNCPoint5[23193] = {X 528.8484, Y 21.2152, Z -7.1667, A 0.000, B 0.000, C 0.000 }
gfCNCPoint5[23194] = {X 529.4646, Y 21.7385, Z -7.1667, A 0.000, B 0.000, C 0.000 }
gfCNCPoint5[23195] = {X 529.9654, Y 22.3729, Z -7.1667, A 0.000, B 0.000, C 0.000 }
gfCNCPoint5[23196] = {X 534.8719, Y 22.3731, Z -7.1667, A 0.000, B 0.000, C 0.000 }
gfCNCPoint5[23197] = {X 534.8719, Y 19.4626, Z -7.1667, A 0.000, B 0.000, C 0.000 }
gfCNCPoint5[23198] = {X 524.0610, Y 19.4625, Z -7.1667, A 0.000, B 0.000, C 0.000 }
gfCNCPoint5[23199] = {X 524.0087, Y 19.5442, Z -7.1667, A 0.000, B 0.000, C 0.000 }
gfCNCPoint5[23200] = {X 523.5061, Y 20.1604, Z -7.1667, A 0.000, B 0.000, C 0.000 }
gfCNCPoint5[23201] = {X 522.8935, Y 20.6674, Z -7.1667, A 0.000, B 0.000, C 0.000 }
gfCNCPoint5[23202] = {X 522.1942, Y 21.0459, Z -7.1667, A 0.000, B 0.000, C 0.000 }
gfCNCPoint5[23203] = {X 521.4348, Y 21.2816, Z -7.1667, A 0.000, B 0.000, C 0.000 }
gfCNCPoint5[23204] = {X 520.6440, Y 21.3656, Z -7.1667, A 0.000, B 0.000, C 0.000 }
gfCNCPoint5[23205] = {X 519.9691, Y 21.3657, Z -7.1667, A 0.000, B 0.000, C 0.000 }
gfCNCPoint5[23206] = {X 519.0612, Y 21.2634, Z -7.1667, A 0.000, B 0.000, C 0.000 }
gfCNCPoint5[23207] = {X 518.1989, Y 20.9617, Z -7.1667, A 0.000, B 0.000, C 0.000 }
gfCNCPoint5[23208] = {X 517.4253, Y 20.4756, Z -7.1667, A 0.000, B 0.000, C 0.000 }
gfCNCPoint5[23209] = {X 516.7792, Y 19.8296, Z -7.1667, A 0.000, B 0.000, C 0.000 }
gfCNCPoint5[23210] = {X 516.2932, Y 19.0560, Z -7.1667, A 0.000, B 0.000, C 0.000 }
gfCNCPoint5[23211] = {X 515.9914, Y 18.1936, Z -7.1667, A 0.000, B 0.000, C 0.000 }
gfCNCPoint5[23212] = {X 515.8891, Y 17.2857, Z -7.1667, A 0.000, B 0.000, C 0.000 }
gfCNCPoint5[23213] = {X 515.8891, Y 10.3077, Z -7.1667, A 0.000, B 0.000, C 0.000 }
gfCNCPoint5[23214] = {X 515.9902, Y 9.4050, Z -7.1667, A 0.000, B 0.000, C 0.000 }
gfCNCPoint5[23215] = {X 516.2885, Y 8.5471, Z -7.1667, A 0.000, B 0.000, C 0.000 }
gfCNCPoint5[23216] = {X 516.7693, Y 7.7764, Z -7.1667, A 0.000, B 0.000, C 0.000 }
gfCNCPoint5[23217] = {X 517.4086, Y 7.1312, Z -7.1667, A 0.000, B 0.000, C 0.000 }
gfCNCPoint5[23218] = {X 518.1749, Y 6.6434, Z -7.1667, A 0.000, B 0.000, C 0.000 }
gfCNCPoint5[23219] = {X 519.0301, Y 6.3372, Z -7.1667, A 0.000, B 0.000, C 0.000 }
gfCNCPoint5[23220] = {X 519.9318, Y 6.2279, Z -7.1667, A 0.000, B 0.000, C 0.000 }
gfCNCPoint5[23221] = {X 520.6480, Y 6.2279, Z -7.1667, A 0.000, B 0.000, C 0.000 }
gfCNCPoint5[23222] = {X 521.4519, Y 6.3153, Z -7.1667, A 0.000, B 0.000, C 0.000 }
gfCNCPoint5[23223] = {X 522.2227, Y 6.5596, Z -7.1667, A 0.000, B 0.000, C 0.000 }
gfCNCPoint5[23224] = {X 522.9303, Y 6.9512, Z -7.1667, A 0.000, B 0.000, C 0.000 }
gfCNCPoint5[23225] = {X 523.5467, Y 7.4746, Z -7.1667, A 0.000, B 0.000, C 0.000 }
gfCNCPoint5[23226] = {X 524.0478, Y 8.1092, Z -7.1667, A 0.000, B 0.000, C 0.000 }
gfCNCPoint5[23227] = {X 533.9633, Y 8.1094, Z -7.1667, A 0.000, B 0.000, C 0.000 }
gfCNCPoint5[23228] = {X 533.9634, Y 4.1094, Z -7.1667, A 0.000, B 0.000, C 0.000 }
gfCNCPoint5[23229] = {X 533.9633, Y 8.1894, Z -7.1667, A 0.000, B 0.000, C 0.000 }
gfCNCPoint5[23230] = {X 543.7544, Y 8.1896, Z -7.1667, A 0.000, B 0.000, C 0.000 }
gfCNCPoint5[23231] = {X 544.6629, Y 8.2679, Z -7.1667, A 0.000, B 0.000, C 0.000 }
gfCNCPoint5[23232] = {X 545.5301, Y 8.5498, Z -7.1667, A 0.000, B 0.000, C 0.000 }
gfCNCPoint5[23233] = {X 546.3111, Y 9.0205, Z -7.1667, A 0.000, B 0.000, C 0.000 }
gfCNCPoint5[23234] = {X 546.9654, Y 9.6557, Z -7.1667, A 0.000, B 0.000, C 0.000 }
gfCNCPoint5[23235] = {X 547.4589, Y 10.4225, Z -7.1667, A 0.000, B 0.000, C 0.000 }
gfCNCPoint5[23236] = {X 547.7663, Y 11.2810, Z -7.1667, A 0.000, B 0.000, C 0.000 }
gfCNCPoint5[23237] = {X 547.8714, Y 12.1868, Z -7.1667, A 0.000, B 0.000, C 0.000 }
gfCNCPoint5[23238] = {X 547.8712, Y 13.0192, Z -7.1667, A 0.000, B 0.000, C 0.000 }
gfCNCPoint5[23239] = {X 547.7627, Y 13.9043, Z -7.1667, A 0.000, B 0.000, C 0.000 }
gfCNCPoint5[23240] = {X 547.4608, Y 14.7433, Z -7.1667, A 0.000, B 0.000, C 0.000 }
gfCNCPoint5[23241] = {X 546.9806, Y 15.4946, Z -7.1667, A 0.000, B 0.000, C 0.000 }
gfCNCPoint5[23242] = {X 546.3458, Y 16.1209, Z -7.1667, A 0.000, B 0.000, C 0.000 }
gfCNCPoint5[23243] = {X 546.3450, Y 41.0654, Z -7.1667, A 0.000, B 0.000, C 0.000 }
gfCNCPoint5[23244] = {X 546.4837, Y 41.1796, Z -7.1667, A 0.000, B 0.000, C 0.000 }
gfCNCPoint5[23245] = {X 547.0694, Y 41.8060, Z -7.1667, A 0.000, B 0.000, C 0.000 }
gfCNCPoint5[23246] = {X 547.5080, Y 42.5429, Z -7.1667, A 0.000, B 0.000, C 0.000 }
gfCNCPoint5[23247] = {X 547.7795, Y 43.3563, Z -7.1667, A 0.000, B 0.000, C 0.000 }
gfCNCPoint5[23248] = {X 547.8714, Y 44.2089, Z -7.1667, A 0.000, B 0.000, C 0.000 }
gfCNCPoint5[23249] = {X 547.8714, Y 45.0000, Z -7.1667, A 0.000, B 0.000, C 0.000 }
gfCNCPoint5[23250] = {X 547.7663, Y 45.9058, Z -7.1667, A 0.000, B 0.000, C 0.000 }
gfCNCPoint5[23251] = {X 547.4589, Y 46.7643, Z -7.1667, A 0.000, B 0.000, C 0.000 }
gfCNCPoint5[23252] = {X 546.9653, Y 47.5310, Z -7.1667, A 0.000, B 0.000, C 0.000 }
gfCNCPoint5[23253] = {X 546.3111, Y 48.1661, Z -7.1667, A 0.000, B 0.000, C 0.000 }
gfCNCPoint5[23254] = {X 545.5301, Y 48.6368, Z -7.1667, A 0.000, B 0.000, C 0.000 }
gfCNCPoint5[23255] = {X 544.6628, Y 48.9186, Z -7.1667, A 0.000, B 0.000, C 0.000 }
gfCNCPoint5[23256] = {X 543.7544, Y 48.9969, Z -7.1667, A 0.000, B 0.000, C 0.000 }
gfCNCPoint5[23257] = {X 523.8765, Y 48.9973, Z -7.1667, A 0.000, B 0.000, C 0.000 }
gfCNCPoint5[23258] = {X 523.3701, Y 49.6283, Z -7.1667, A 0.000, B 0.000, C 0.000 }
gfCNCPoint5[23259] = {X 522.7510, Y 50.1492, Z -7.1667, A 0.000, B 0.000, C 0.000 }
gfCNCPoint5[23260] = {X 522.0426, Y 50.5403, Z -7.1667, A 0.000, B 0.000, C 0.000 }
gfCNCPoint5[23261] = {X 521.2720, Y 50.7867, Z -7.1667, A 0.000, B 0.000, C 0.000 }
gfCNCPoint5[23262] = {X 520.4681, Y 50.8791, Z -7.1667, A 0.000, B 0.000, C 0.000 }
gfCNCPoint5[23263] = {X 519.7998, Y 50.8791, Z -7.1667, A 0.000, B 0.000, C 0.000 }
gfCNCPoint5[23264] = {X 518.9097, Y 50.7788, Z -7.1667, A 0.000, B 0.000, C 0.000 }
gfCNCPoint5[23265] = {X 518.0642, Y 50.4830, Z -7.1667, A 0.000, B 0.000, C 0.000 }
gfCNCPoint5[23266] = {X 517.3058, Y 50.0064, Z -7.1667, A 0.000, B 0.000, C 0.000 }
gfCNCPoint5[23267] = {X 516.6724, Y 49.3731, Z -7.1667, A 0.000, B 0.000, C 0.000 }
gfCNCPoint5[23268] = {X 516.1959, Y 48.6147, Z -7.1667, A 0.000, B 0.000, C 0.000 }
gfCNCPoint5[23269] = {X 515.9001, Y 47.7692, Z -7.1667, A 0.000, B 0.000, C 0.000 }
gfCNCPoint5[23270] = {X 515.7998, Y 46.8791, Z -7.1667, A 0.000, B 0.000, C 0.000 }
gfCNCPoint5[23271] = {X 515.7998, Y 39.9011, Z -7.1667, A 0.000, B 0.000, C 0.000 }
gfCNCPoint5[23272] = {X 515.9001, Y 39.0110, Z -7.1667, A 0.000, B 0.000, C 0.000 }
gfCNCPoint5[23273] = {X 516.1959, Y 38.1656, Z -7.1667, A 0.000, B 0.000, C 0.000 }
gfCNCPoint5[23274] = {X 516.6725, Y 37.4071, Z -7.1667, A 0.000, B 0.000, C 0.000 }
gfCNCPoint5[23275] = {X 517.3058, Y 36.7738, Z -7.1667, A 0.000, B 0.000, C 0.000 }
gfCNCPoint5[23276] = {X 518.0643, Y 36.2972, Z -7.1667, A 0.000, B 0.000, C 0.000 }
gfCNCPoint5[23277] = {X 518.9097, Y 36.0014, Z -7.1667, A 0.000, B 0.000, C 0.000 }
gfCNCPoint5[23278] = {X 519.7998, Y 35.9011, Z -7.1667, A 0.000, B 0.000, C 0.000 }
gfCNCPoint5[23279] = {X 520.5225, Y 35.9015, Z -7.1667, A 0.000, B 0.000, C 0.000 }
gfCNCPoint5[23280] = {X 521.3204, Y 35.9929, Z -7.1667, A 0.000, B 0.000, C 0.000 }
gfCNCPoint5[23281] = {X 522.0839, Y 36.2419, Z -7.1667, A 0.000, B 0.000, C 0.000 }
gfCNCPoint5[23282] = {X 522.7823, Y 36.6385, Z -7.1667, A 0.000, B 0.000, C 0.000 }
gfCNCPoint5[23283] = {X 523.3874, Y 37.1665, Z -7.1667, A 0.000, B 0.000, C 0.000 }
gfCNCPoint5[23284] = {X 523.8748, Y 37.8048, Z -7.1667, A 0.000, B 0.000, C 0.000 }
gfCNCPoint5[23285] = {X 534.9519, Y 37.8051, Z -7.1667, A 0.000, B 0.000, C 0.000 }
gfCNCPoint5[23286] = {X 534.9519, Y 33.6462, Z -7.1667, A 0.000, B 0.000, C 0.000 }
gfCNCPoint5[23287] = {X 529.9338, Y 33.6460, Z -7.1667, A 0.000, B 0.000, C 0.000 }
gfCNCPoint5[23288] = {X 529.8222, Y 33.8190, Z -7.1667, A 0.000, B 0.000, C 0.000 }
gfCNCPoint5[23289] = {X 529.1827, Y 34.5419, Z -7.1667, A 0.000, B 0.000, C 0.000 }
gfCNCPoint5[23290] = {X 528.3887, Y 35.0905, Z -7.1667, A 0.000, B 0.000, C 0.000 }
gfCNCPoint5[23291] = {X 527.4864, Y 35.4330, Z -7.1667, A 0.000, B 0.000, C 0.000 }
gfCNCPoint5[23292] = {X 526.5283, Y 35.5495, Z -7.1667, A 0.000, B 0.000, C 0.000 }
gfCNCPoint5[23293] = {X 525.8868, Y 35.5495, Z -7.1667, A 0.000, B 0.000, C 0.000 }
gfCNCPoint5[23294] = {X 524.9967, Y 35.4492, Z -7.1667, A 0.000, B 0.000, C 0.000 }
gfCNCPoint5[23295] = {X 524.1512, Y 35.1533, Z -7.1667, A 0.000, B 0.000, C 0.000 }
gfCNCPoint5[23296] = {X 523.3928, Y 34.6768, Z -7.1667, A 0.000, B 0.000, C 0.000 }
gfCNCPoint5[23297] = {X 522.7594, Y 34.0434, Z -7.1667, A 0.000, B 0.000, C 0.000 }
gfCNCPoint5[23298] = {X 522.2829, Y 33.2850, Z -7.1667, A 0.000, B 0.000, C 0.000 }
gfCNCPoint5[23299] = {X 521.9870, Y 32.4395, Z -7.1667, A 0.000, B 0.000, C 0.000 }
gfCNCPoint5[23300] = {X 521.8868, Y 31.5495, Z -7.1667, A 0.000, B 0.000, C 0.000 }
gfCNCPoint5[23301] = {X 521.8868, Y 24.5714, Z -7.1667, A 0.000, B 0.000, C 0.000 }
gfCNCPoint5[23302] = {X 521.9870, Y 23.6813, Z -7.1667, A 0.000, B 0.000, C 0.000 }
gfCNCPoint5[23303] = {X 522.2829, Y 22.8359, Z -7.1667, A 0.000, B 0.000, C 0.000 }
gfCNCPoint5[23304] = {X 522.7594, Y 22.0775, Z -7.1667, A 0.000, B 0.000, C 0.000 }
gfCNCPoint5[23305] = {X 523.3928, Y 21.4441, Z -7.1667, A 0.000, B 0.000, C 0.000 }
gfCNCPoint5[23306] = {X 524.1512, Y 20.9675, Z -7.1667, A 0.000, B 0.000, C 0.000 }
gfCNCPoint5[23307] = {X 524.9967, Y 20.6717, Z -7.1667, A 0.000, B 0.000, C 0.000 }
gfCNCPoint5[23308] = {X 525.8868, Y 20.5714, Z -7.1667, A 0.000, B 0.000, C 0.000 }
gfCNCPoint5[23309] = {X 526.5664, Y 20.5716, Z -7.1667, A 0.000, B 0.000, C 0.000 }
gfCNCPoint5[23310] = {X 527.3628, Y 20.6594, Z -7.1667, A 0.000, B 0.000, C 0.000 }
gfCNCPoint5[23311] = {X 528.1256, Y 20.9041, Z -7.1667, A 0.000, B 0.000, C 0.000 }
gfCNCPoint5[23312] = {X 528.8244, Y 21.2960, Z -7.1667, A 0.000, B 0.000, C 0.000 }
gfCNCPoint5[23313] = {X 529.4311, Y 21.8193, Z -7.1667, A 0.000, B 0.000, C 0.000 }
gfCNCPoint5[23314] = {X 529.9214, Y 22.4529, Z -7.1667, A 0.000, B 0.000, C 0.000 }
gfCNCPoint5[23315] = {X 534.9519, Y 22.4531, Z -7.1667, A 0.000, B 0.000, C 0.000 }
gfCNCPoint5[23316] = {X 534.9519, Y 19.3826, Z -7.1667, A 0.000, B 0.000, C 0.000 }
gfCNCPoint5[23317] = {X 524.0172, Y 19.3825, Z -7.1667, A 0.000, B 0.000, C 0.000 }
gfCNCPoint5[23318] = {X 523.9044, Y 19.5555, Z -7.1667, A 0.000, B 0.000, C 0.000 }
gfCNCPoint5[23319] = {X 523.2650, Y 20.2783, Z -7.1667, A 0.000, B 0.000, C 0.000 }
gfCNCPoint5[23320] = {X 522.4710, Y 20.8268, Z -7.1667, A 0.000, B 0.000, C 0.000 }
gfCNCPoint5[23321] = {X 521.5687, Y 21.1693, Z -7.1667, A 0.000, B 0.000, C 0.000 }
gfCNCPoint5[23322] = {X 520.6107, Y 21.2857, Z -7.1667, A 0.000, B 0.000, C 0.000 }
gfCNCPoint5[23323] = {X 519.9691, Y 21.2857, Z -7.1667, A 0.000, B 0.000, C 0.000 }
gfCNCPoint5[23324] = {X 519.0790, Y 21.1854, Z -7.1667, A 0.000, B 0.000, C 0.000 }
gfCNCPoint5[23325] = {X 518.2336, Y 20.8896, Z -7.1667, A 0.000, B 0.000, C 0.000 }
gfCNCPoint5[23326] = {X 517.4751, Y 20.4130, Z -7.1667, A 0.000, B 0.000, C 0.000 }
gfCNCPoint5[23327] = {X 516.8418, Y 19.7797, Z -7.1667, A 0.000, B 0.000, C 0.000 }
gfCNCPoint5[23328] = {X 516.3652, Y 19.0212, Z -7.1667, A 0.000, B 0.000, C 0.000 }
gfCNCPoint5[23329] = {X 516.0694, Y 18.1758, Z -7.1667, A 0.000, B 0.000, C 0.000 }
gfCNCPoint5[23330] = {X 515.9691, Y 17.2857, Z -7.1667, A 0.000, B 0.000, C 0.000 }
gfCNCPoint5[23331] = {X 515.9691, Y 10.3077, Z -7.1667, A 0.000, B 0.000, C 0.000 }
gfCNCPoint5[23332] = {X 516.0694, Y 9.4176, Z -7.1667, A 0.000, B 0.000, C 0.000 }
gfCNCPoint5[23333] = {X 516.3652, Y 8.5721, Z -7.1667, A 0.000, B 0.000, C 0.000 }
gfCNCPoint5[23334] = {X 516.8418, Y 7.8137, Z -7.1667, A 0.000, B 0.000, C 0.000 }
gfCNCPoint5[23335] = {X 517.4752, Y 7.1803, Z -7.1667, A 0.000, B 0.000, C 0.000 }
gfCNCPoint5[23336] = {X 518.2336, Y 6.7038, Z -7.1667, A 0.000, B 0.000, C 0.000 }
gfCNCPoint5[23337] = {X 519.0791, Y 6.4080, Z -7.1667, A 0.000, B 0.000, C 0.000 }
gfCNCPoint5[23338] = {X 519.9692, Y 6.3077, Z -7.1667, A 0.000, B 0.000, C 0.000 }
gfCNCPoint5[23339] = {X 520.6472, Y 6.3079, Z -7.1667, A 0.000, B 0.000, C 0.000 }
gfCNCPoint5[23340] = {X 521.4439, Y 6.3954, Z -7.1667, A 0.000, B 0.000, C 0.000 }
gfCNCPoint5[23341] = {X 522.2072, Y 6.6401, Z -7.1667, A 0.000, B 0.000, C 0.000 }
gfCNCPoint5[23342] = {X 522.9063, Y 7.0319, Z -7.1667, A 0.000, B 0.000, C 0.000 }
gfCNCPoint5[23343] = {X 523.5133, Y 7.5553, Z -7.1667, A 0.000, B 0.000, C 0.000 }
gfCNCPoint5[23344] = {X 524.0037, Y 8.1892, Z -7.1667, A 0.000, B 0.000, C 0.000 }
gfCNCPoint5[23345] = {X 533.9633, Y 8.1894, Z -7.1667, A 0.000, B 0.000, C 0.000 }
gfCNCPoint5[23346] = {X 533.9634, Y 4.1094, Z -7.1667, A 0.000, B 0.000, C 0.000 }
gfCNCPoint5[23347] = {X 533.9634, Y 4.1094, Z -4.1667, A 0.000, B 0.000, C 0.000 }
gfCNCPoint5[23348] = {X 533.9634, Y 4.1094, Z 11.0000, A 0.000, B 0.000, C 0.000 }
gfCNCPoint5[23349] = {X 419.6150, Y 26.5282, Z 11.0000, A 0.000, B 0.000, C 0.000 }
gfCNCPoint5[23350] = {X 419.6150, Y 26.5282, Z -4.1667, A 0.000, B 0.000, C 0.000 }
gfCNCPoint5[23351] = {X 419.6150, Y 26.5282, Z -7.1667, A 0.000, B 0.000, C 0.000 }
gfCNCPoint5[23352] = {X 416.1514, Y 24.3717, Z -7.1667, A 0.000, B 0.000, C 0.000 }
gfCNCPoint5[23353] = {X 411.5479, Y 31.7654, Z -7.1667, A 0.000, B 0.000, C 0.000 }
gfCNCPoint5[23354] = {X 411.5485, Y 40.8975, Z -7.1667, A 0.000, B 0.000, C 0.000 }
gfCNCPoint5[23355] = {X 412.1867, Y 41.5834, Z -7.1667, A 0.000, B 0.000, C 0.000 }
gfCNCPoint5[23356] = {X 412.6667, Y 42.3879, Z -7.1667, A 0.000, B 0.000, C 0.000 }
gfCNCPoint5[23357] = {X 412.9672, Y 43.2752, Z -7.1667, A 0.000, B 0.000, C 0.000 }
gfCNCPoint5[23358] = {X 413.0747, Y 44.2059, Z -7.1667, A 0.000, B 0.000, C 0.000 }
gfCNCPoint5[23359] = {X 413.0745, Y 45.0415, Z -7.1667, A 0.000, B 0.000, C 0.000 }
gfCNCPoint5[23360] = {X 412.9583, Y 45.9960, Z -7.1667, A 0.000, B 0.000, C 0.000 }
gfCNCPoint5[23361] = {X 412.6339, Y 46.9011, Z -7.1667, A 0.000, B 0.000, C 0.000 }
gfCNCPoint5[23362] = {X 412.1173, Y 47.7120, Z -7.1667, A 0.000, B 0.000, C 0.000 }
gfCNCPoint5[23363] = {X 411.4342, Y 48.3886, Z -7.1667, A 0.000, B 0.000, C 0.000 }
gfCNCPoint5[23364] = {X 410.6184, Y 48.8973, Z -7.1667, A 0.000, B 0.000, C 0.000 }
gfCNCPoint5[23365] = {X 409.7102, Y 49.2130, Z -7.1667, A 0.000, B 0.000, C 0.000 }
gfCNCPoint5[23366] = {X 408.7547, Y 49.3200, Z -7.1667, A 0.000, B 0.000, C 0.000 }
gfCNCPoint5[23367] = {X 402.3112, Y 49.3200, Z -7.1667, A 0.000, B 0.000, C 0.000 }
gfCNCPoint5[23368] = {X 401.3546, Y 49.2127, Z -7.1667, A 0.000, B 0.000, C 0.000 }
gfCNCPoint5[23369] = {X 400.4455, Y 48.8963, Z -7.1667, A 0.000, B 0.000, C 0.000 }
gfCNCPoint5[23370] = {X 399.6290, Y 48.3864, Z -7.1667, A 0.000, B 0.000, C 0.000 }
gfCNCPoint5[23371] = {X 398.9457, Y 47.7084, Z -7.1667, A 0.000, B 0.000, C 0.000 }
gfCNCPoint5[23372] = {X 398.4295, Y 46.8959, Z -7.1667, A 0.000, B 0.000, C 0.000 }
gfCNCPoint5[23373] = {X 398.1060, Y 45.9892, Z -7.1667, A 0.000, B 0.000, C 0.000 }
gfCNCPoint5[23374] = {X 397.9913, Y 45.0335, Z -7.1667, A 0.000, B 0.000, C 0.000 }
gfCNCPoint5[23375] = {X 397.9916, Y 44.1528, Z -7.1667, A 0.000, B 0.000, C 0.000 }
gfCNCPoint5[23376] = {X 398.1015, Y 43.2391, Z -7.1667, A 0.000, B 0.000, C 0.000 }
gfCNCPoint5[23377] = {X 398.4024, Y 42.3694, Z -7.1667, A 0.000, B 0.000, C 0.000 }
gfCNCPoint5[23378] = {X 398.8807, Y 41.5832, Z -7.1667, A 0.000, B 0.000, C 0.000 }
gfCNCPoint5[23379] = {X 399.5147, Y 40.9161, Z -7.1667, A 0.000, B 0.000, C 0.000 }
gfCNCPoint5[23380] = {X 399.4729, Y 31.6023, Z -7.1667, A 0.000, B 0.000, C 0.000 }
gfCNCPoint5[23381] = {X 393.4355, Y 21.1034, Z -7.1667, A 0.000, B 0.000, C 0.000 }
gfCNCPoint5[23382] = {X 392.5862, Y 19.6600, Z -7.1667, A 0.000, B 0.000, C 0.000 }
gfCNCPoint5[23383] = {X 391.7081, Y 18.2340, Z -7.1667, A 0.000, B 0.000, C 0.000 }
gfCNCPoint5[23384] = {X 391.2272, Y 17.5669, Z -7.1667, A 0.000, B 0.000, C 0.000 }
gfCNCPoint5[23385] = {X 390.6667, Y 16.9651, Z -7.1667, A 0.000, B 0.000, C 0.000 }
gfCNCPoint5[23386] = {X 389.7900, Y 16.4727, Z -7.1667, A 0.000, B 0.000, C 0.000 }
gfCNCPoint5[23387] = {X 389.0510, Y 15.7910, Z -7.1667, A 0.000, B 0.000, C 0.000 }
gfCNCPoint5[23388] = {X 388.4895, Y 14.9569, Z -7.1667, A 0.000, B 0.000, C 0.000 }
gfCNCPoint5[23389] = {X 388.1361, Y 14.0156, Z -7.1667, A 0.000, B 0.000, C 0.000 }
gfCNCPoint5[23390] = {X 388.0098, Y 13.0180, Z -7.1667, A 0.000, B 0.000, C 0.000 }
gfCNCPoint5[23391] = {X 388.0096, Y 12.1868, Z -7.1667, A 0.000, B 0.000, C 0.000 }
gfCNCPoint5[23392] = {X 388.1179, Y 11.2255, Z -7.1667, A 0.000, B 0.000, C 0.000 }
gfCNCPoint5[23393] = {X 388.4374, Y 10.3125, Z -7.1667, A 0.000, B 0.000, C 0.000 }
gfCNCPoint5[23394] = {X 388.9521, Y 9.4933, Z -7.1667, A 0.000, B 0.000, C 0.000 }
gfCNCPoint5[23395] = {X 389.6361, Y 8.8093, Z -7.1667, A 0.000, B 0.000, C 0.000 }
gfCNCPoint5[23396] = {X 390.4552, Y 8.2946, Z -7.1667, A 0.000, B 0.000, C 0.000 }
gfCNCPoint5[23397] = {X 391.3683, Y 7.9751, Z -7.1667, A 0.000, B 0.000, C 0.000 }
gfCNCPoint5[23398] = {X 392.3296, Y 7.8668, Z -7.1667, A 0.000, B 0.000, C 0.000 }
gfCNCPoint5[23399] = {X 399.1118, Y 7.8668, Z -7.1667, A 0.000, B 0.000, C 0.000 }
gfCNCPoint5[23400] = {X 400.0730, Y 7.9751, Z -7.1667, A 0.000, B 0.000, C 0.000 }
gfCNCPoint5[23401] = {X 400.9861, Y 8.2946, Z -7.1667, A 0.000, B 0.000, C 0.000 }
gfCNCPoint5[23402] = {X 401.8052, Y 8.8093, Z -7.1667, A 0.000, B 0.000, C 0.000 }
gfCNCPoint5[23403] = {X 402.4893, Y 9.4933, Z -7.1667, A 0.000, B 0.000, C 0.000 }
gfCNCPoint5[23404] = {X 403.0039, Y 10.3124, Z -7.1667, A 0.000, B 0.000, C 0.000 }
gfCNCPoint5[23405] = {X 403.3234, Y 11.2255, Z -7.1667, A 0.000, B 0.000, C 0.000 }
gfCNCPoint5[23406] = {X 403.4318, Y 12.1868, Z -7.1667, A 0.000, B 0.000, C 0.000 }
gfCNCPoint5[23407] = {X 403.4318, Y 12.9782, Z -7.1667, A 0.000, B 0.000, C 0.000 }
gfCNCPoint5[23408] = {X 403.3293, Y 13.9134, Z -7.1667, A 0.000, B 0.000, C 0.000 }
gfCNCPoint5[23409] = {X 403.0267, Y 14.8044, Z -7.1667, A 0.000, B 0.000, C 0.000 }
gfCNCPoint5[23410] = {X 405.3556, Y 18.8224, Z -7.1667, A 0.000, B 0.000, C 0.000 }
gfCNCPoint5[23411] = {X 407.8731, Y 14.7532, Z -7.1667, A 0.000, B 0.000, C 0.000 }
gfCNCPoint5[23412] = {X 407.5920, Y 13.9040, Z -7.1667, A 0.000, B 0.000, C 0.000 }
gfCNCPoint5[23413] = {X 407.4917, Y 13.0151, Z -7.1667, A 0.000, B 0.000, C 0.000 }
gfCNCPoint5[23414] = {X 407.4915, Y 12.1868, Z -7.1667, A 0.000, B 0.000, C 0.000 }
gfCNCPoint5[23415] = {X 407.5999, Y 11.2255, Z -7.1667, A 0.000, B 0.000, C 0.000 }
gfCNCPoint5[23416] = {X 407.9194, Y 10.3124, Z -7.1667, A 0.000, B 0.000, C 0.000 }
gfCNCPoint5[23417] = {X 408.4340, Y 9.4933, Z -7.1667, A 0.000, B 0.000, C 0.000 }
gfCNCPoint5[23418] = {X 409.1181, Y 8.8093, Z -7.1667, A 0.000, B 0.000, C 0.000 }
gfCNCPoint5[23419] = {X 409.9372, Y 8.2946, Z -7.1667, A 0.000, B 0.000, C 0.000 }
gfCNCPoint5[23420] = {X 410.8502, Y 7.9751, Z -7.1667, A 0.000, B 0.000, C 0.000 }
gfCNCPoint5[23421] = {X 411.8115, Y 7.8668, Z -7.1667, A 0.000, B 0.000, C 0.000 }
gfCNCPoint5[23422] = {X 419.3245, Y 7.8668, Z -7.1667, A 0.000, B 0.000, C 0.000 }
gfCNCPoint5[23423] = {X 420.2858, Y 7.9751, Z -7.1667, A 0.000, B 0.000, C 0.000 }
gfCNCPoint5[23424] = {X 421.1988, Y 8.2946, Z -7.1667, A 0.000, B 0.000, C 0.000 }
gfCNCPoint5[23425] = {X 422.0179, Y 8.8093, Z -7.1667, A 0.000, B 0.000, C 0.000 }
gfCNCPoint5[23426] = {X 422.7020, Y 9.4933, Z -7.1667, A 0.000, B 0.000, C 0.000 }
gfCNCPoint5[23427] = {X 423.2166, Y 10.3124, Z -7.1667, A 0.000, B 0.000, C 0.000 }
gfCNCPoint5[23428] = {X 423.5361, Y 11.2255, Z -7.1667, A 0.000, B 0.000, C 0.000 }
gfCNCPoint5[23429] = {X 423.6445, Y 12.1868, Z -7.1667, A 0.000, B 0.000, C 0.000 }
gfCNCPoint5[23430] = {X 423.6445, Y 12.9801, Z -7.1667, A 0.000, B 0.000, C 0.000 }
gfCNCPoint5[23431] = {X 423.5520, Y 13.8467, Z -7.1667, A 0.000, B 0.000, C 0.000 }
gfCNCPoint5[23432] = {X 423.2898, Y 14.6779, Z -7.1667, A 0.000, B 0.000, C 0.000 }
gfCNCPoint5[23433] = {X 422.8683, Y 15.4407, Z -7.1667, A 0.000, B 0.000, C 0.000 }
gfCNCPoint5[23434] = {X 422.3041, Y 16.1049, Z -7.1667, A 0.000, B 0.000, C 0.000 }
gfCNCPoint5[23435] = {X 421.6196, Y 16.6444, Z -7.1667, A 0.000, B 0.000, C 0.000 }
gfCNCPoint5[23436] = {X 420.8418, Y 17.0376, Z -7.1667, A 0.000, B 0.000, C 0.000 }
gfCNCPoint5[23437] = {X 420.1254, Y 18.0009, Z -7.1667, A 0.000, B 0.000, C 0.000 }
gfCNCPoint5[23438] = {X 419.4772, Y 19.0115, Z -7.1667, A 0.000, B 0.000, C 0.000 }
gfCNCPoint5[23439] = {X 417.9942, Y 21.4120, Z -7.1667, A 0.000, B 0.000, C 0.000 }
gfCNCPoint5[23440] = {X 416.1514, Y 24.3717, Z -7.1667, A 0.000, B 0.000, C 0.000 }
gfCNCPoint5[23441] = {X 419.5470, Y 26.4859, Z -7.1667, A 0.000, B 0.000, C 0.000 }
gfCNCPoint5[23442] = {X 416.0835, Y 24.3294, Z -7.1667, A 0.000, B 0.000, C 0.000 }
gfCNCPoint5[23443] = {X 411.4679, Y 31.7425, Z -7.1667, A 0.000, B 0.000, C 0.000 }
gfCNCPoint5[23444] = {X 411.4685, Y 40.9342, Z -7.1667, A 0.000, B 0.000, C 0.000 }
gfCNCPoint5[23445] = {X 412.1063, Y 41.6097, Z -7.1667, A 0.000, B 0.000, C 0.000 }
gfCNCPoint5[23446] = {X 412.5864, Y 42.4049, Z -7.1667, A 0.000, B 0.000, C 0.000 }
gfCNCPoint5[23447] = {X 412.8871, Y 43.2839, Z -7.1667, A 0.000, B 0.000, C 0.000 }
gfCNCPoint5[23448] = {X 412.9947, Y 44.2066, Z -7.1667, A 0.000, B 0.000, C 0.000 }
gfCNCPoint5[23449] = {X 412.9945, Y 45.0408, Z -7.1667, A 0.000, B 0.000, C 0.000 }
gfCNCPoint5[23450] = {X 412.8805, Y 45.9775, Z -7.1667, A 0.000, B 0.000, C 0.000 }
gfCNCPoint5[23451] = {X 412.5621, Y 46.8659, Z -7.1667, A 0.000, B 0.000, C 0.000 }
gfCNCPoint5[23452] = {X 412.0551, Y 47.6618, Z -7.1667, A 0.000, B 0.000, C 0.000 }
gfCNCPoint5[23453] = {X 411.3846, Y 48.3258, Z -7.1667, A 0.000, B 0.000, C 0.000 }
gfCNCPoint5[23454] = {X 410.5838, Y 48.8251, Z -7.1667, A 0.000, B 0.000, C 0.000 }
gfCNCPoint5[23455] = {X 409.6925, Y 49.1350, Z -7.1667, A 0.000, B 0.000, C 0.000 }
gfCNCPoint5[23456] = {X 408.7547, Y 49.2400, Z -7.1667, A 0.000, B 0.000, C 0.000 }
gfCNCPoint5[23457] = {X 402.3112, Y 49.2400, Z -7.1667, A 0.000, B 0.000, C 0.000 }
gfCNCPoint5[23458] = {X 401.3723, Y 49.1347, Z -7.1667, A 0.000, B 0.000, C 0.000 }
gfCNCPoint5[23459] = {X 400.4800, Y 48.8242, Z -7.1667, A 0.000, B 0.000, C 0.000 }
gfCNCPoint5[23460] = {X 399.6786, Y 48.3237, Z -7.1667, A 0.000, B 0.000, C 0.000 }
gfCNCPoint5[23461] = {X 399.0080, Y 47.6582, Z -7.1667, A 0.000, B 0.000, C 0.000 }
gfCNCPoint5[23462] = {X 398.5013, Y 46.8608, Z -7.1667, A 0.000, B 0.000, C 0.000 }
gfCNCPoint5[23463] = {X 398.1839, Y 45.9709, Z -7.1667, A 0.000, B 0.000, C 0.000 }
gfCNCPoint5[23464] = {X 398.0713, Y 45.0329, Z -7.1667, A 0.000, B 0.000, C 0.000 }
gfCNCPoint5[23465] = {X 398.0716, Y 44.1538, Z -7.1667, A 0.000, B 0.000, C 0.000 }
gfCNCPoint5[23466] = {X 398.1815, Y 43.2480, Z -7.1667, A 0.000, B 0.000, C 0.000 }
gfCNCPoint5[23467] = {X 398.4827, Y 42.3867, Z -7.1667, A 0.000, B 0.000, C 0.000 }
gfCNCPoint5[23468] = {X 398.9612, Y 41.6098, Z -7.1667, A 0.000, B 0.000, C 0.000 }
gfCNCPoint5[23469] = {X 399.5948, Y 40.9532, Z -7.1667, A 0.000, B 0.000, C 0.000 }
gfCNCPoint5[23470] = {X 399.5528, Y 31.5808, Z -7.1667, A 0.000, B 0.000, C 0.000 }
gfCNCPoint5[23471] = {X 393.5049, Y 21.0635, Z -7.1667, A 0.000, B 0.000, C 0.000 }
gfCNCPoint5[23472] = {X 392.6547, Y 19.6188, Z -7.1667, A 0.000, B 0.000, C 0.000 }
gfCNCPoint5[23473] = {X 391.7758, Y 18.1914, Z -7.1667, A 0.000, B 0.000, C 0.000 }
gfCNCPoint5[23474] = {X 391.2844, Y 17.5104, Z -7.1667, A 0.000, B 0.000, C 0.000 }
gfCNCPoint5[23475] = {X 390.7110, Y 16.8969, Z -7.1667, A 0.000, B 0.000, C 0.000 }
gfCNCPoint5[23476] = {X 389.8465, Y 16.4148, Z -7.1667, A 0.000, B 0.000, C 0.000 }
gfCNCPoint5[23477] = {X 389.1174, Y 15.7455, Z -7.1667, A 0.000, B 0.000, C 0.000 }
gfCNCPoint5[23478] = {X 388.5633, Y 14.9254, Z -7.1667, A 0.000, B 0.000, C 0.000 }
gfCNCPoint5[23479] = {X 388.2144, Y 13.9992, Z -7.1667, A 0.000, B 0.000, C 0.000 }
gfCNCPoint5[23480] = {X 388.0898, Y 13.0173, Z -7.1667, A 0.000, B 0.000, C 0.000 }
gfCNCPoint5[23481] = {X 388.0896, Y 12.1868, Z -7.1667, A 0.000, B 0.000, C 0.000 }
gfCNCPoint5[23482] = {X 388.1959, Y 11.2433, Z -7.1667, A 0.000, B 0.000, C 0.000 }
gfCNCPoint5[23483] = {X 388.5095, Y 10.3472, Z -7.1667, A 0.000, B 0.000, C 0.000 }
gfCNCPoint5[23484] = {X 389.0147, Y 9.5432, Z -7.1667, A 0.000, B 0.000, C 0.000 }
gfCNCPoint5[23485] = {X 389.6860, Y 8.8719, Z -7.1667, A 0.000, B 0.000, C 0.000 }
gfCNCPoint5[23486] = {X 390.4900, Y 8.3667, Z -7.1667, A 0.000, B 0.000, C 0.000 }
gfCNCPoint5[23487] = {X 391.3861, Y 8.0531, Z -7.1667, A 0.000, B 0.000, C 0.000 }
gfCNCPoint5[23488] = {X 392.3296, Y 7.9468, Z -7.1667, A 0.000, B 0.000, C 0.000 }
gfCNCPoint5[23489] = {X 399.1118, Y 7.9468, Z -7.1667, A 0.000, B 0.000, C 0.000 }
gfCNCPoint5[23490] = {X 400.0552, Y 8.0531, Z -7.1667, A 0.000, B 0.000, C 0.000 }
gfCNCPoint5[23491] = {X 400.9514, Y 8.3667, Z -7.1667, A 0.000, B 0.000, C 0.000 }
gfCNCPoint5[23492] = {X 401.7554, Y 8.8718, Z -7.1667, A 0.000, B 0.000, C 0.000 }
gfCNCPoint5[23493] = {X 402.4267, Y 9.5432, Z -7.1667, A 0.000, B 0.000, C 0.000 }
gfCNCPoint5[23494] = {X 402.9319, Y 10.3471, Z -7.1667, A 0.000, B 0.000, C 0.000 }
gfCNCPoint5[23495] = {X 403.2455, Y 11.2433, Z -7.1667, A 0.000, B 0.000, C 0.000 }
gfCNCPoint5[23496] = {X 403.3518, Y 12.1868, Z -7.1667, A 0.000, B 0.000, C 0.000 }
gfCNCPoint5[23497] = {X 403.3518, Y 12.9782, Z -7.1667, A 0.000, B 0.000, C 0.000 }
gfCNCPoint5[23498] = {X 403.2466, Y 13.9164, Z -7.1667, A 0.000, B 0.000, C 0.000 }
gfCNCPoint5[23499] = {X 402.9364, Y 14.8081, Z -7.1667, A 0.000, B 0.000, C 0.000 }
gfCNCPoint5[23500] = {X 405.3534, Y 18.9781, Z -7.1667, A 0.000, B 0.000, C 0.000 }
gfCNCPoint5[23501] = {X 407.9637, Y 14.7589, Z -7.1667, A 0.000, B 0.000, C 0.000 }
gfCNCPoint5[23502] = {X 407.6747, Y 13.9076, Z -7.1667, A 0.000, B 0.000, C 0.000 }
gfCNCPoint5[23503] = {X 407.5717, Y 13.0144, Z -7.1667, A 0.000, B 0.000, C 0.000 }
gfCNCPoint5[23504] = {X 407.5715, Y 12.1868, Z -7.1667, A 0.000, B 0.000, C 0.000 }
gfCNCPoint5[23505] = {X 407.6778, Y 11.2433, Z -7.1667, A 0.000, B 0.000, C 0.000 }
gfCNCPoint5[23506] = {X 407.9914, Y 10.3471, Z -7.1667, A 0.000, B 0.000, C 0.000 }
gfCNCPoint5[23507] = {X 408.4966, Y 9.5432, Z -7.1667, A 0.000, B 0.000, C 0.000 }
gfCNCPoint5[23508] = {X 409.1679, Y 8.8718, Z -7.1667, A 0.000, B 0.000, C 0.000 }
gfCNCPoint5[23509] = {X 409.9719, Y 8.3667, Z -7.1667, A 0.000, B 0.000, C 0.000 }
gfCNCPoint5[23510] = {X 410.8680, Y 8.0531, Z -7.1667, A 0.000, B 0.000, C 0.000 }
gfCNCPoint5[23511] = {X 411.8115, Y 7.9468, Z -7.1667, A 0.000, B 0.000, C 0.000 }
gfCNCPoint5[23512] = {X 419.3245, Y 7.9468, Z -7.1667, A 0.000, B 0.000, C 0.000 }
gfCNCPoint5[23513] = {X 420.2679, Y 8.0531, Z -7.1667, A 0.000, B 0.000, C 0.000 }
gfCNCPoint5[23514] = {X 421.1641, Y 8.3667, Z -7.1667, A 0.000, B 0.000, C 0.000 }
gfCNCPoint5[23515] = {X 421.9681, Y 8.8718, Z -7.1667, A 0.000, B 0.000, C 0.000 }
gfCNCPoint5[23516] = {X 422.6394, Y 9.5432, Z -7.1667, A 0.000, B 0.000, C 0.000 }
gfCNCPoint5[23517] = {X 423.1446, Y 10.3471, Z -7.1667, A 0.000, B 0.000, C 0.000 }
gfCNCPoint5[23518] = {X 423.4582, Y 11.2433, Z -7.1667, A 0.000, B 0.000, C 0.000 }
gfCNCPoint5[23519] = {X 423.5645, Y 12.1868, Z -7.1667, A 0.000, B 0.000, C 0.000 }
gfCNCPoint5[23520] = {X 423.5645, Y 12.9796, Z -7.1667, A 0.000, B 0.000, C 0.000 }
gfCNCPoint5[23521] = {X 423.4730, Y 13.8339, Z -7.1667, A 0.000, B 0.000, C 0.000 }
gfCNCPoint5[23522] = {X 423.2135, Y 14.6529, Z -7.1667, A 0.000, B 0.000, C 0.000 }
gfCNCPoint5[23523] = {X 422.7964, Y 15.4041, Z -7.1667, A 0.000, B 0.000, C 0.000 }
gfCNCPoint5[23524] = {X 422.2382, Y 16.0573, Z -7.1667, A 0.000, B 0.000, C 0.000 }
gfCNCPoint5[23525] = {X 421.5614, Y 16.5865, Z -7.1667, A 0.000, B 0.000, C 0.000 }
gfCNCPoint5[23526] = {X 420.7929, Y 16.9707, Z -7.1667, A 0.000, B 0.000, C 0.000 }
gfCNCPoint5[23527] = {X 420.0660, Y 17.9462, Z -7.1667, A 0.000, B 0.000, C 0.000 }
gfCNCPoint5[23528] = {X 419.4088, Y 18.9700, Z -7.1667, A 0.000, B 0.000, C 0.000 }
gfCNCPoint5[23529] = {X 417.9262, Y 21.3699, Z -7.1667, A 0.000, B 0.000, C 0.000 }
gfCNCPoint5[23530] = {X 416.0835, Y 24.3294, Z -7.1667, A 0.000, B 0.000, C 0.000 }
gfCNCPoint5[23531] = {X 419.4791, Y 26.4436, Z -7.1667, A 0.000, B 0.000, C 0.000 }
gfCNCPoint5[23532] = {X 416.0156, Y 24.2871, Z -7.1667, A 0.000, B 0.000, C 0.000 }
gfCNCPoint5[23533] = {X 411.3879, Y 31.7196, Z -7.1667, A 0.000, B 0.000, C 0.000 }
gfCNCPoint5[23534] = {X 411.3885, Y 40.9713, Z -7.1667, A 0.000, B 0.000, C 0.000 }
gfCNCPoint5[23535] = {X 412.0259, Y 41.6362, Z -7.1667, A 0.000, B 0.000, C 0.000 }
gfCNCPoint5[23536] = {X 412.5061, Y 42.4221, Z -7.1667, A 0.000, B 0.000, C 0.000 }
gfCNCPoint5[23537] = {X 412.8070, Y 43.2926, Z -7.1667, A 0.000, B 0.000, C 0.000 }
gfCNCPoint5[23538] = {X 412.9147, Y 44.2074, Z -7.1667, A 0.000, B 0.000, C 0.000 }
gfCNCPoint5[23539] = {X 412.9145, Y 45.0400, Z -7.1667, A 0.000, B 0.000, C 0.000 }
gfCNCPoint5[23540] = {X 412.8026, Y 45.9591, Z -7.1667, A 0.000, B 0.000, C 0.000 }
gfCNCPoint5[23541] = {X 412.4902, Y 46.8306, Z -7.1667, A 0.000, B 0.000, C 0.000 }
gfCNCPoint5[23542] = {X 411.9928, Y 47.6115, Z -7.1667, A 0.000, B 0.000, C 0.000 }
gfCNCPoint5[23543] = {X 411.3350, Y 48.2631, Z -7.1667, A 0.000, B 0.000, C 0.000 }
gfCNCPoint5[23544] = {X 410.5493, Y 48.7530, Z -7.1667, A 0.000, B 0.000, C 0.000 }
gfCNCPoint5[23545] = {X 409.6748, Y 49.0570, Z -7.1667, A 0.000, B 0.000, C 0.000 }
gfCNCPoint5[23546] = {X 408.7547, Y 49.1600, Z -7.1667, A 0.000, B 0.000, C 0.000 }
gfCNCPoint5[23547] = {X 402.3112, Y 49.1600, Z -7.1667, A 0.000, B 0.000, C 0.000 }
gfCNCPoint5[23548] = {X 401.3900, Y 49.0567, Z -7.1667, A 0.000, B 0.000, C 0.000 }
gfCNCPoint5[23549] = {X 400.5146, Y 48.7520, Z -7.1667, A 0.000, B 0.000, C 0.000 }
gfCNCPoint5[23550] = {X 399.7283, Y 48.2610, Z -7.1667, A 0.000, B 0.000, C 0.000 }
gfCNCPoint5[23551] = {X 399.0703, Y 47.6081, Z -7.1667, A 0.000, B 0.000, C 0.000 }
gfCNCPoint5[23552] = {X 398.5732, Y 46.8257, Z -7.1667, A 0.000, B 0.000, C 0.000 }
gfCNCPoint5[23553] = {X 398.2617, Y 45.9526, Z -7.1667, A 0.000, B 0.000, C 0.000 }
gfCNCPoint5[23554] = {X 398.1513, Y 45.0322, Z -7.1667, A 0.000, B 0.000, C 0.000 }
gfCNCPoint5[23555] = {X 398.1516, Y 44.1549, Z -7.1667, A 0.000, B 0.000, C 0.000 }
gfCNCPoint5[23556] = {X 398.2616, Y 43.2570, Z -7.1667, A 0.000, B 0.000, C 0.000 }
gfCNCPoint5[23557] = {X 398.5630, Y 42.4041, Z -7.1667, A 0.000, B 0.000, C 0.000 }
gfCNCPoint5[23558] = {X 399.0417, Y 41.6366, Z -7.1667, A 0.000, B 0.000, C 0.000 }
gfCNCPoint5[23559] = {X 399.6750, Y 40.9907, Z -7.1667, A 0.000, B 0.000, C 0.000 }
gfCNCPoint5[23560] = {X 399.6327, Y 31.5592, Z -7.1667, A 0.000, B 0.000, C 0.000 }
gfCNCPoint5[23561] = {X 393.5742, Y 21.0236, Z -7.1667, A 0.000, B 0.000, C 0.000 }
gfCNCPoint5[23562] = {X 392.7233, Y 19.5775, Z -7.1667, A 0.000, B 0.000, C 0.000 }
gfCNCPoint5[23563] = {X 391.8435, Y 18.1487, Z -7.1667, A 0.000, B 0.000, C 0.000 }
gfCNCPoint5[23564] = {X 391.3414, Y 17.4539, Z -7.1667, A 0.000, B 0.000, C 0.000 }
gfCNCPoint5[23565] = {X 390.7550, Y 16.8285, Z -7.1667, A 0.000, B 0.000, C 0.000 }
gfCNCPoint5[23566] = {X 389.9029, Y 16.3568, Z -7.1667, A 0.000, B 0.000, C 0.000 }
gfCNCPoint5[23567] = {X 389.1837, Y 15.7000, Z -7.1667, A 0.000, B 0.000, C 0.000 }
gfCNCPoint5[23568] = {X 388.6370, Y 14.8939, Z -7.1667, A 0.000, B 0.000, C 0.000 }
gfCNCPoint5[23569] = {X 388.2928, Y 13.9828, Z -7.1667, A 0.000, B 0.000, C 0.000 }
gfCNCPoint5[23570] = {X 388.1698, Y 13.0166, Z -7.1667, A 0.000, B 0.000, C 0.000 }
gfCNCPoint5[23571] = {X 388.1696, Y 12.1868, Z -7.1667, A 0.000, B 0.000, C 0.000 }
gfCNCPoint5[23572] = {X 388.2739, Y 11.2611, Z -7.1667, A 0.000, B 0.000, C 0.000 }
gfCNCPoint5[23573] = {X 388.5816, Y 10.3819, Z -7.1667, A 0.000, B 0.000, C 0.000 }
gfCNCPoint5[23574] = {X 389.0772, Y 9.5931, Z -7.1667, A 0.000, B 0.000, C 0.000 }
gfCNCPoint5[23575] = {X 389.7359, Y 8.9344, Z -7.1667, A 0.000, B 0.000, C 0.000 }
gfCNCPoint5[23576] = {X 390.5247, Y 8.4388, Z -7.1667, A 0.000, B 0.000, C 0.000 }
gfCNCPoint5[23577] = {X 391.4039, Y 8.1311, Z -7.1667, A 0.000, B 0.000, C 0.000 }
gfCNCPoint5[23578] = {X 392.3296, Y 8.0268, Z -7.1667, A 0.000, B 0.000, C 0.000 }
gfCNCPoint5[23579] = {X 399.1118, Y 8.0268, Z -7.1667, A 0.000, B 0.000, C 0.000 }
gfCNCPoint5[23580] = {X 400.0374, Y 8.1311, Z -7.1667, A 0.000, B 0.000, C 0.000 }
gfCNCPoint5[23581] = {X 400.9167, Y 8.4388, Z -7.1667, A 0.000, B 0.000, C 0.000 }
gfCNCPoint5[23582] = {X 401.7055, Y 8.9344, Z -7.1667, A 0.000, B 0.000, C 0.000 }
gfCNCPoint5[23583] = {X 402.3642, Y 9.5931, Z -7.1667, A 0.000, B 0.000, C 0.000 }
gfCNCPoint5[23584] = {X 402.8598, Y 10.3819, Z -7.1667, A 0.000, B 0.000, C 0.000 }
gfCNCPoint5[23585] = {X 403.1675, Y 11.2611, Z -7.1667, A 0.000, B 0.000, C 0.000 }
gfCNCPoint5[23586] = {X 403.2718, Y 12.1868, Z -7.1667, A 0.000, B 0.000, C 0.000 }
gfCNCPoint5[23587] = {X 403.2718, Y 12.9782, Z -7.1667, A 0.000, B 0.000, C 0.000 }
gfCNCPoint5[23588] = {X 403.1639, Y 13.9192, Z -7.1667, A 0.000, B 0.000, C 0.000 }
gfCNCPoint5[23589] = {X 402.8459, Y 14.8115, Z -7.1667, A 0.000, B 0.000, C 0.000 }
gfCNCPoint5[23590] = {X 405.3512, Y 19.1338, Z -7.1667, A 0.000, B 0.000, C 0.000 }
gfCNCPoint5[23591] = {X 408.0545, Y 14.7642, Z -7.1667, A 0.000, B 0.000, C 0.000 }
gfCNCPoint5[23592] = {X 407.7575, Y 13.9110, Z -7.1667, A 0.000, B 0.000, C 0.000 }
gfCNCPoint5[23593] = {X 407.6517, Y 13.0137, Z -7.1667, A 0.000, B 0.000, C 0.000 }
gfCNCPoint5[23594] = {X 407.6515, Y 12.1868, Z -7.1667, A 0.000, B 0.000, C 0.000 }
gfCNCPoint5[23595] = {X 407.7558, Y 11.2611, Z -7.1667, A 0.000, B 0.000, C 0.000 }
gfCNCPoint5[23596] = {X 408.0635, Y 10.3819, Z -7.1667, A 0.000, B 0.000, C 0.000 }
gfCNCPoint5[23597] = {X 408.5591, Y 9.5931, Z -7.1667, A 0.000, B 0.000, C 0.000 }
gfCNCPoint5[23598] = {X 409.2178, Y 8.9344, Z -7.1667, A 0.000, B 0.000, C 0.000 }
gfCNCPoint5[23599] = {X 410.0066, Y 8.4388, Z -7.1667, A 0.000, B 0.000, C 0.000 }
gfCNCPoint5[23600] = {X 410.8859, Y 8.1311, Z -7.1667, A 0.000, B 0.000, C 0.000 }
gfCNCPoint5[23601] = {X 411.8115, Y 8.0268, Z -7.1667, A 0.000, B 0.000, C 0.000 }
gfCNCPoint5[23602] = {X 419.3245, Y 8.0268, Z -7.1667, A 0.000, B 0.000, C 0.000 }
gfCNCPoint5[23603] = {X 420.2501, Y 8.1311, Z -7.1667, A 0.000, B 0.000, C 0.000 }
gfCNCPoint5[23604] = {X 421.1294, Y 8.4388, Z -7.1667, A 0.000, B 0.000, C 0.000 }
gfCNCPoint5[23605] = {X 421.9182, Y 8.9344, Z -7.1667, A 0.000, B 0.000, C 0.000 }
gfCNCPoint5[23606] = {X 422.5769, Y 9.5931, Z -7.1667, A 0.000, B 0.000, C 0.000 }
gfCNCPoint5[23607] = {X 423.0725, Y 10.3819, Z -7.1667, A 0.000, B 0.000, C 0.000 }
gfCNCPoint5[23608] = {X 423.3802, Y 11.2611, Z -7.1667, A 0.000, B 0.000, C 0.000 }
gfCNCPoint5[23609] = {X 423.4845, Y 12.1868, Z -7.1667, A 0.000, B 0.000, C 0.000 }
gfCNCPoint5[23610] = {X 423.4845, Y 12.9791, Z -7.1667, A 0.000, B 0.000, C 0.000 }
gfCNCPoint5[23611] = {X 423.3939, Y 13.8210, Z -7.1667, A 0.000, B 0.000, C 0.000 }
gfCNCPoint5[23612] = {X 423.1371, Y 14.6279, Z -7.1667, A 0.000, B 0.000, C 0.000 }
gfCNCPoint5[23613] = {X 422.7244, Y 15.3673, Z -7.1667, A 0.000, B 0.000, C 0.000 }
gfCNCPoint5[23614] = {X 422.1725, Y 16.0095, Z -7.1667, A 0.000, B 0.000, C 0.000 }
gfCNCPoint5[23615] = {X 421.5034, Y 16.5285, Z -7.1667, A 0.000, B 0.000, C 0.000 }
gfCNCPoint5[23616] = {X 420.7442, Y 16.9036, Z -7.1667, A 0.000, B 0.000, C 0.000 }
gfCNCPoint5[23617] = {X 420.0066, Y 17.8914, Z -7.1667, A 0.000, B 0.000, C 0.000 }
gfCNCPoint5[23618] = {X 419.3404, Y 18.9286, Z -7.1667, A 0.000, B 0.000, C 0.000 }
gfCNCPoint5[23619] = {X 417.8582, Y 21.3277, Z -7.1667, A 0.000, B 0.000, C 0.000 }
gfCNCPoint5[23620] = {X 416.0156, Y 24.2871, Z -7.1667, A 0.000, B 0.000, C 0.000 }
gfCNCPoint5[23621] = {X 419.4112, Y 26.4013, Z -7.1667, A 0.000, B 0.000, C 0.000 }
gfCNCPoint5[23622] = {X 415.9477, Y 24.2448, Z -7.1667, A 0.000, B 0.000, C 0.000 }
gfCNCPoint5[23623] = {X 411.3079, Y 31.6968, Z -7.1667, A 0.000, B 0.000, C 0.000 }
gfCNCPoint5[23624] = {X 411.3085, Y 41.0088, Z -7.1667, A 0.000, B 0.000, C 0.000 }
gfCNCPoint5[23625] = {X 411.9454, Y 41.6630, Z -7.1667, A 0.000, B 0.000, C 0.000 }
gfCNCPoint5[23626] = {X 412.4258, Y 42.4395, Z -7.1667, A 0.000, B 0.000, C 0.000 }
gfCNCPoint5[23627] = {X 412.7270, Y 43.3014, Z -7.1667, A 0.000, B 0.000, C 0.000 }
gfCNCPoint5[23628] = {X 412.8347, Y 44.2081, Z -7.1667, A 0.000, B 0.000, C 0.000 }
gfCNCPoint5[23629] = {X 412.8345, Y 45.0392, Z -7.1667, A 0.000, B 0.000, C 0.000 }
gfCNCPoint5[23630] = {X 412.7248, Y 45.9406, Z -7.1667, A 0.000, B 0.000, C 0.000 }
gfCNCPoint5[23631] = {X 412.4184, Y 46.7954, Z -7.1667, A 0.000, B 0.000, C 0.000 }
gfCNCPoint5[23632] = {X 411.9305, Y 47.5613, Z -7.1667, A 0.000, B 0.000, C 0.000 }
gfCNCPoint5[23633] = {X 411.2854, Y 48.2003, Z -7.1667, A 0.000, B 0.000, C 0.000 }
gfCNCPoint5[23634] = {X 410.5148, Y 48.6808, Z -7.1667, A 0.000, B 0.000, C 0.000 }
gfCNCPoint5[23635] = {X 409.6571, Y 48.9789, Z -7.1667, A 0.000, B 0.000, C 0.000 }
gfCNCPoint5[23636] = {X 408.7547, Y 49.0800, Z -7.1667, A 0.000, B 0.000, C 0.000 }
gfCNCPoint5[23637] = {X 402.3112, Y 49.0800, Z -7.1667, A 0.000, B 0.000, C 0.000 }
gfCNCPoint5[23638] = {X 401.4077, Y 48.9787, Z -7.1667, A 0.000, B 0.000, C 0.000 }
gfCNCPoint5[23639] = {X 400.5491, Y 48.6799, Z -7.1667, A 0.000, B 0.000, C 0.000 }
gfCNCPoint5[23640] = {X 399.7780, Y 48.1983, Z -7.1667, A 0.000, B 0.000, C 0.000 }
gfCNCPoint5[23641] = {X 399.1326, Y 47.5579, Z -7.1667, A 0.000, B 0.000, C 0.000 }
gfCNCPoint5[23642] = {X 398.6451, Y 46.7906, Z -7.1667, A 0.000, B 0.000, C 0.000 }
gfCNCPoint5[23643] = {X 398.3396, Y 45.9343, Z -7.1667, A 0.000, B 0.000, C 0.000 }
gfCNCPoint5[23644] = {X 398.2313, Y 45.0316, Z -7.1667, A 0.000, B 0.000, C 0.000 }
gfCNCPoint5[23645] = {X 398.2316, Y 44.1559, Z -7.1667, A 0.000, B 0.000, C 0.000 }
gfCNCPoint5[23646] = {X 398.3416, Y 43.2661, Z -7.1667, A 0.000, B 0.000, C 0.000 }
gfCNCPoint5[23647] = {X 398.6434, Y 42.4218, Z -7.1667, A 0.000, B 0.000, C 0.000 }
gfCNCPoint5[23648] = {X 399.1223, Y 41.6638, Z -7.1667, A 0.000, B 0.000, C 0.000 }
gfCNCPoint5[23649] = {X 399.7552, Y 41.0287, Z -7.1667, A 0.000, B 0.000, C 0.000 }
gfCNCPoint5[23650] = {X 399.7126, Y 31.5377, Z -7.1667, A 0.000, B 0.000, C 0.000 }
gfCNCPoint5[23651] = {X 393.6436, Y 20.9837, Z -7.1667, A 0.000, B 0.000, C 0.000 }
gfCNCPoint5[23652] = {X 392.7918, Y 19.5363, Z -7.1667, A 0.000, B 0.000, C 0.000 }
gfCNCPoint5[23653] = {X 391.9112, Y 18.1061, Z -7.1667, A 0.000, B 0.000, C 0.000 }
gfCNCPoint5[23654] = {X 391.3984, Y 17.3972, Z -7.1667, A 0.000, B 0.000, C 0.000 }
gfCNCPoint5[23655] = {X 390.7989, Y 16.7600, Z -7.1667, A 0.000, B 0.000, C 0.000 }
gfCNCPoint5[23656] = {X 389.9591, Y 16.2987, Z -7.1667, A 0.000, B 0.000, C 0.000 }
gfCNCPoint5[23657] = {X 389.2500, Y 15.6543, Z -7.1667, A 0.000, B 0.000, C 0.000 }
gfCNCPoint5[23658] = {X 388.7108, Y 14.8622, Z -7.1667, A 0.000, B 0.000, C 0.000 }
gfCNCPoint5[23659] = {X 388.3711, Y 13.9663, Z -7.1667, A 0.000, B 0.000, C 0.000 }
gfCNCPoint5[23660] = {X 388.2498, Y 13.0158, Z -7.1667, A 0.000, B 0.000, C 0.000 }
gfCNCPoint5[23661] = {X 388.2496, Y 12.1868, Z -7.1667, A 0.000, B 0.000, C 0.000 }
gfCNCPoint5[23662] = {X 388.3519, Y 11.2789, Z -7.1667, A 0.000, B 0.000, C 0.000 }
gfCNCPoint5[23663] = {X 388.6537, Y 10.4166, Z -7.1667, A 0.000, B 0.000, C 0.000 }
gfCNCPoint5[23664] = {X 389.1398, Y 9.6430, Z -7.1667, A 0.000, B 0.000, C 0.000 }
gfCNCPoint5[23665] = {X 389.7858, Y 8.9969, Z -7.1667, A 0.000, B 0.000, C 0.000 }
gfCNCPoint5[23666] = {X 390.5594, Y 8.5109, Z -7.1667, A 0.000, B 0.000, C 0.000 }
gfCNCPoint5[23667] = {X 391.4217, Y 8.2091, Z -7.1667, A 0.000, B 0.000, C 0.000 }
gfCNCPoint5[23668] = {X 392.3296, Y 8.1068, Z -7.1667, A 0.000, B 0.000, C 0.000 }
gfCNCPoint5[23669] = {X 399.1118, Y 8.1068, Z -7.1667, A 0.000, B 0.000, C 0.000 }
gfCNCPoint5[23670] = {X 400.0196, Y 8.2091, Z -7.1667, A 0.000, B 0.000, C 0.000 }
gfCNCPoint5[23671] = {X 400.8820, Y 8.5109, Z -7.1667, A 0.000, B 0.000, C 0.000 }
gfCNCPoint5[23672] = {X 401.6556, Y 8.9969, Z -7.1667, A 0.000, B 0.000, C 0.000 }
gfCNCPoint5[23673] = {X 402.3016, Y 9.6430, Z -7.1667, A 0.000, B 0.000, C 0.000 }
gfCNCPoint5[23674] = {X 402.7877, Y 10.4166, Z -7.1667, A 0.000, B 0.000, C 0.000 }
gfCNCPoint5[23675] = {X 403.0895, Y 11.2789, Z -7.1667, A 0.000, B 0.000, C 0.000 }
gfCNCPoint5[23676] = {X 403.1918, Y 12.1868, Z -7.1667, A 0.000, B 0.000, C 0.000 }
gfCNCPoint5[23677] = {X 403.1918, Y 12.9782, Z -7.1667, A 0.000, B 0.000, C 0.000 }
gfCNCPoint5[23678] = {X 403.0811, Y 13.9219, Z -7.1667, A 0.000, B 0.000, C 0.000 }
gfCNCPoint5[23679] = {X 402.7551, Y 14.8144, Z -7.1667, A 0.000, B 0.000, C 0.000 }
gfCNCPoint5[23680] = {X 405.3489, Y 19.2894, Z -7.1667, A 0.000, B 0.000, C 0.000 }
gfCNCPoint5[23681] = {X 408.1456, Y 14.7690, Z -7.1667, A 0.000, B 0.000, C 0.000 }
gfCNCPoint5[23682] = {X 408.1088, Y 14.6916, Z -7.1667, A 0.000, B 0.000, C 0.000 }
gfCNCPoint5[23683] = {X 408.0737, Y 14.6135, Z -7.1667, A 0.000, B 0.000, C 0.000 }
gfCNCPoint5[23684] = {X 407.8216, Y 13.8306, Z -7.1667, A 0.000, B 0.000, C 0.000 }
gfCNCPoint5[23685] = {X 407.7317, Y 13.0131, Z -7.1667, A 0.000, B 0.000, C 0.000 }
gfCNCPoint5[23686] = {X 407.7315, Y 12.1868, Z -7.1667, A 0.000, B 0.000, C 0.000 }
gfCNCPoint5[23687] = {X 407.8338, Y 11.2789, Z -7.1667, A 0.000, B 0.000, C 0.000 }
gfCNCPoint5[23688] = {X 408.1356, Y 10.4166, Z -7.1667, A 0.000, B 0.000, C 0.000 }
gfCNCPoint5[23689] = {X 408.6217, Y 9.6430, Z -7.1667, A 0.000, B 0.000, C 0.000 }
gfCNCPoint5[23690] = {X 409.2677, Y 8.9969, Z -7.1667, A 0.000, B 0.000, C 0.000 }
gfCNCPoint5[23691] = {X 410.0413, Y 8.5109, Z -7.1667, A 0.000, B 0.000, C 0.000 }
gfCNCPoint5[23692] = {X 410.9037, Y 8.2091, Z -7.1667, A 0.000, B 0.000, C 0.000 }
gfCNCPoint5[23693] = {X 411.8115, Y 8.1068, Z -7.1667, A 0.000, B 0.000, C 0.000 }
gfCNCPoint5[23694] = {X 419.3245, Y 8.1068, Z -7.1667, A 0.000, B 0.000, C 0.000 }
gfCNCPoint5[23695] = {X 420.2323, Y 8.2091, Z -7.1667, A 0.000, B 0.000, C 0.000 }
gfCNCPoint5[23696] = {X 421.0947, Y 8.5109, Z -7.1667, A 0.000, B 0.000, C 0.000 }
gfCNCPoint5[23697] = {X 421.8683, Y 8.9969, Z -7.1667, A 0.000, B 0.000, C 0.000 }
gfCNCPoint5[23698] = {X 422.5143, Y 9.6430, Z -7.1667, A 0.000, B 0.000, C 0.000 }
gfCNCPoint5[23699] = {X 423.0004, Y 10.4166, Z -7.1667, A 0.000, B 0.000, C 0.000 }
gfCNCPoint5[23700] = {X 423.3022, Y 11.2789, Z -7.1667, A 0.000, B 0.000, C 0.000 }
gfCNCPoint5[23701] = {X 423.4045, Y 12.1868, Z -7.1667, A 0.000, B 0.000, C 0.000 }
gfCNCPoint5[23702] = {X 423.4045, Y 12.9785, Z -7.1667, A 0.000, B 0.000, C 0.000 }
gfCNCPoint5[23703] = {X 423.3149, Y 13.8081, Z -7.1667, A 0.000, B 0.000, C 0.000 }
gfCNCPoint5[23704] = {X 423.0608, Y 14.6028, Z -7.1667, A 0.000, B 0.000, C 0.000 }
gfCNCPoint5[23705] = {X 422.6526, Y 15.3305, Z -7.1667, A 0.000, B 0.000, C 0.000 }
gfCNCPoint5[23706] = {X 422.1068, Y 15.9615, Z -7.1667, A 0.000, B 0.000, C 0.000 }
gfCNCPoint5[23707] = {X 421.4455, Y 16.4703, Z -7.1667, A 0.000, B 0.000, C 0.000 }
gfCNCPoint5[23708] = {X 420.6957, Y 16.8363, Z -7.1667, A 0.000, B 0.000, C 0.000 }
gfCNCPoint5[23709] = {X 419.9474, Y 17.8364, Z -7.1667, A 0.000, B 0.000, C 0.000 }
gfCNCPoint5[23710] = {X 419.2719, Y 18.8871, Z -7.1667, A 0.000, B 0.000, C 0.000 }
gfCNCPoint5[23711] = {X 417.7903, Y 21.2855, Z -7.1667, A 0.000, B 0.000, C 0.000 }
gfCNCPoint5[23712] = {X 415.9477, Y 24.2448, Z -7.1667, A 0.000, B 0.000, C 0.000 }
gfCNCPoint5[23713] = {X 419.3433, Y 26.3591, Z -7.1667, A 0.000, B 0.000, C 0.000 }
gfCNCPoint5[23714] = {X 415.8798, Y 24.2026, Z -7.1667, A 0.000, B 0.000, C 0.000 }
gfCNCPoint5[23715] = {X 411.2279, Y 31.6739, Z -7.1667, A 0.000, B 0.000, C 0.000 }
gfCNCPoint5[23716] = {X 411.2285, Y 41.0467, Z -7.1667, A 0.000, B 0.000, C 0.000 }
gfCNCPoint5[23717] = {X 411.8650, Y 41.6901, Z -7.1667, A 0.000, B 0.000, C 0.000 }
gfCNCPoint5[23718] = {X 412.3455, Y 42.4570, Z -7.1667, A 0.000, B 0.000, C 0.000 }
gfCNCPoint5[23719] = {X 412.6469, Y 43.3103, Z -7.1667, A 0.000, B 0.000, C 0.000 }
gfCNCPoint5[23720] = {X 412.7547, Y 44.2088, Z -7.1667, A 0.000, B 0.000, C 0.000 }
gfCNCPoint5[23721] = {X 412.7545, Y 45.0384, Z -7.1667, A 0.000, B 0.000, C 0.000 }
gfCNCPoint5[23722] = {X 412.6469, Y 45.9222, Z -7.1667, A 0.000, B 0.000, C 0.000 }
gfCNCPoint5[23723] = {X 412.3466, Y 46.7602, Z -7.1667, A 0.000, B 0.000, C 0.000 }
gfCNCPoint5[23724] = {X 411.8683, Y 47.5111, Z -7.1667, A 0.000, B 0.000, C 0.000 }
gfCNCPoint5[23725] = {X 411.2357, Y 48.1376, Z -7.1667, A 0.000, B 0.000, C 0.000 }
gfCNCPoint5[23726] = {X 410.4803, Y 48.6086, Z -7.1667, A 0.000, B 0.000, C 0.000 }
gfCNCPoint5[23727] = {X 409.6394, Y 48.9009, Z -7.1667, A 0.000, B 0.000, C 0.000 }
gfCNCPoint5[23728] = {X 408.7547, Y 49.0000, Z -7.1667, A 0.000, B 0.000, C 0.000 }
gfCNCPoint5[23729] = {X 402.3112, Y 49.0000, Z -7.1667, A 0.000, B 0.000, C 0.000 }
gfCNCPoint5[23730] = {X 401.4211, Y 48.8997, Z -7.1667, A 0.000, B 0.000, C 0.000 }
gfCNCPoint5[23731] = {X 400.5757, Y 48.6039, Z -7.1667, A 0.000, B 0.000, C 0.000 }
gfCNCPoint5[23732] = {X 399.8172, Y 48.1273, Z -7.1667, A 0.000, B 0.000, C 0.000 }
gfCNCPoint5[23733] = {X 399.1839, Y 47.4939, Z -7.1667, A 0.000, B 0.000, C 0.000 }
gfCNCPoint5[23734] = {X 398.7073, Y 46.7355, Z -7.1667, A 0.000, B 0.000, C 0.000 }
gfCNCPoint5[23735] = {X 398.4115, Y 45.8901, Z -7.1667, A 0.000, B 0.000, C 0.000 }
gfCNCPoint5[23736] = {X 398.3112, Y 45.0000, Z -7.1667, A 0.000, B 0.000, C 0.000 }
gfCNCPoint5[23737] = {X 398.3115, Y 44.1569, Z -7.1667, A 0.000, B 0.000, C 0.000 }
gfCNCPoint5[23738] = {X 398.4217, Y 43.2753, Z -7.1667, A 0.000, B 0.000, C 0.000 }
gfCNCPoint5[23739] = {X 398.7237, Y 42.4397, Z -7.1667, A 0.000, B 0.000, C 0.000 }
gfCNCPoint5[23740] = {X 399.2028, Y 41.6913, Z -7.1667, A 0.000, B 0.000, C 0.000 }
gfCNCPoint5[23741] = {X 399.8352, Y 41.0672, Z -7.1667, A 0.000, B 0.000, C 0.000 }
gfCNCPoint5[23742] = {X 399.8364, Y 31.5925, Z -7.1667, A 0.000, B 0.000, C 0.000 }
gfCNCPoint5[23743] = {X 393.7129, Y 20.9439, Z -7.1667, A 0.000, B 0.000, C 0.000 }
gfCNCPoint5[23744] = {X 392.8604, Y 19.4950, Z -7.1667, A 0.000, B 0.000, C 0.000 }
gfCNCPoint5[23745] = {X 391.9789, Y 18.0635, Z -7.1667, A 0.000, B 0.000, C 0.000 }
gfCNCPoint5[23746] = {X 391.4553, Y 17.3405, Z -7.1667, A 0.000, B 0.000, C 0.000 }
gfCNCPoint5[23747] = {X 390.8426, Y 16.6913, Z -7.1667, A 0.000, B 0.000, C 0.000 }
gfCNCPoint5[23748] = {X 390.0091, Y 16.2361, Z -7.1667, A 0.000, B 0.000, C 0.000 }
gfCNCPoint5[23749] = {X 389.3064, Y 15.5972, Z -7.1667, A 0.000, B 0.000, C 0.000 }
gfCNCPoint5[23750] = {X 388.7742, Y 14.8107, Z -7.1667, A 0.000, B 0.000, C 0.000 }
gfCNCPoint5[23751] = {X 388.4424, Y 13.9209, Z -7.1667, A 0.000, B 0.000, C 0.000 }
gfCNCPoint5[23752] = {X 388.3296, Y 12.9780, Z -7.1667, A 0.000, B 0.000, C 0.000 }
gfCNCPoint5[23753] = {X 388.3296, Y 12.1868, Z -7.1667, A 0.000, B 0.000, C 0.000 }
gfCNCPoint5[23754] = {X 388.4299, Y 11.2967, Z -7.1667, A 0.000, B 0.000, C 0.000 }
gfCNCPoint5[23755] = {X 388.7258, Y 10.4513, Z -7.1667, A 0.000, B 0.000, C 0.000 }
gfCNCPoint5[23756] = {X 389.2023, Y 9.6929, Z -7.1667, A 0.000, B 0.000, C 0.000 }
gfCNCPoint5[23757] = {X 389.8357, Y 9.0595, Z -7.1667, A 0.000, B 0.000, C 0.000 }
gfCNCPoint5[23758] = {X 390.5941, Y 8.5829, Z -7.1667, A 0.000, B 0.000, C 0.000 }
gfCNCPoint5[23759] = {X 391.4395, Y 8.2871, Z -7.1667, A 0.000, B 0.000, C 0.000 }
gfCNCPoint5[23760] = {X 392.3296, Y 8.1868, Z -7.1667, A 0.000, B 0.000, C 0.000 }
gfCNCPoint5[23761] = {X 399.1118, Y 8.1868, Z -7.1667, A 0.000, B 0.000, C 0.000 }
gfCNCPoint5[23762] = {X 400.0018, Y 8.2871, Z -7.1667, A 0.000, B 0.000, C 0.000 }
gfCNCPoint5[23763] = {X 400.8473, Y 8.5829, Z -7.1667, A 0.000, B 0.000, C 0.000 }
gfCNCPoint5[23764] = {X 401.6057, Y 9.0595, Z -7.1667, A 0.000, B 0.000, C 0.000 }
gfCNCPoint5[23765] = {X 402.2391, Y 9.6929, Z -7.1667, A 0.000, B 0.000, C 0.000 }
gfCNCPoint5[23766] = {X 402.7156, Y 10.4513, Z -7.1667, A 0.000, B 0.000, C 0.000 }
gfCNCPoint5[23767] = {X 403.0115, Y 11.2967, Z -7.1667, A 0.000, B 0.000, C 0.000 }
gfCNCPoint5[23768] = {X 403.1118, Y 12.1868, Z -7.1667, A 0.000, B 0.000, C 0.000 }
gfCNCPoint5[23769] = {X 403.1115, Y 13.0192, Z -7.1667, A 0.000, B 0.000, C 0.000 }
gfCNCPoint5[23770] = {X 402.9933, Y 13.9442, Z -7.1667, A 0.000, B 0.000, C 0.000 }
gfCNCPoint5[23771] = {X 402.6641, Y 14.8167, Z -7.1667, A 0.000, B 0.000, C 0.000 }
gfCNCPoint5[23772] = {X 405.2576, Y 19.3199, Z -7.1667, A 0.000, B 0.000, C 0.000 }
gfCNCPoint5[23773] = {X 405.3703, Y 19.4071, Z -7.1667, A 0.000, B 0.000, C 0.000 }
gfCNCPoint5[23774] = {X 408.1936, Y 14.8341, Z -7.1667, A 0.000, B 0.000, C 0.000 }
gfCNCPoint5[23775] = {X 408.2428, Y 14.7847, Z -7.1667, A 0.000, B 0.000, C 0.000 }
gfCNCPoint5[23776] = {X 408.1935, Y 14.6838, Z -7.1667, A 0.000, B 0.000, C 0.000 }
gfCNCPoint5[23777] = {X 408.1470, Y 14.5815, Z -7.1667, A 0.000, B 0.000, C 0.000 }
gfCNCPoint5[23778] = {X 407.8963, Y 13.7971, Z -7.1667, A 0.000, B 0.000, C 0.000 }
gfCNCPoint5[23779] = {X 407.8115, Y 12.9780, Z -7.1667, A 0.000, B 0.000, C 0.000 }
gfCNCPoint5[23780] = {X 407.8115, Y 12.1868, Z -7.1667, A 0.000, B 0.000, C 0.000 }
gfCNCPoint5[23781] = {X 407.9118, Y 11.2967, Z -7.1667, A 0.000, B 0.000, C 0.000 }
gfCNCPoint5[23782] = {X 408.2077, Y 10.4513, Z -7.1667, A 0.000, B 0.000, C 0.000 }
gfCNCPoint5[23783] = {X 408.6842, Y 9.6929, Z -7.1667, A 0.000, B 0.000, C 0.000 }
gfCNCPoint5[23784] = {X 409.3176, Y 9.0595, Z -7.1667, A 0.000, B 0.000, C 0.000 }
gfCNCPoint5[23785] = {X 410.0760, Y 8.5829, Z -7.1667, A 0.000, B 0.000, C 0.000 }
gfCNCPoint5[23786] = {X 410.9215, Y 8.2871, Z -7.1667, A 0.000, B 0.000, C 0.000 }
gfCNCPoint5[23787] = {X 411.8115, Y 8.1868, Z -7.1667, A 0.000, B 0.000, C 0.000 }
gfCNCPoint5[23788] = {X 419.3245, Y 8.1868, Z -7.1667, A 0.000, B 0.000, C 0.000 }
gfCNCPoint5[23789] = {X 420.2145, Y 8.2871, Z -7.1667, A 0.000, B 0.000, C 0.000 }
gfCNCPoint5[23790] = {X 421.0600, Y 8.5829, Z -7.1667, A 0.000, B 0.000, C 0.000 }
gfCNCPoint5[23791] = {X 421.8184, Y 9.0595, Z -7.1667, A 0.000, B 0.000, C 0.000 }
gfCNCPoint5[23792] = {X 422.4518, Y 9.6929, Z -7.1667, A 0.000, B 0.000, C 0.000 }
gfCNCPoint5[23793] = {X 422.9283, Y 10.4513, Z -7.1667, A 0.000, B 0.000, C 0.000 }
gfCNCPoint5[23794] = {X 423.2242, Y 11.2967, Z -7.1667, A 0.000, B 0.000, C 0.000 }
gfCNCPoint5[23795] = {X 423.3245, Y 12.1868, Z -7.1667, A 0.000, B 0.000, C 0.000 }
gfCNCPoint5[23796] = {X 423.3245, Y 12.9780, Z -7.1667, A 0.000, B 0.000, C 0.000 }
gfCNCPoint5[23797] = {X 423.2359, Y 13.7951, Z -7.1667, A 0.000, B 0.000, C 0.000 }
gfCNCPoint5[23798] = {X 422.9845, Y 14.5776, Z -7.1667, A 0.000, B 0.000, C 0.000 }
gfCNCPoint5[23799] = {X 422.5808, Y 15.2935, Z -7.1667, A 0.000, B 0.000, C 0.000 }
gfCNCPoint5[23800] = {X 422.0412, Y 15.9134, Z -7.1667, A 0.000, B 0.000, C 0.000 }
gfCNCPoint5[23801] = {X 421.3877, Y 16.4120, Z -7.1667, A 0.000, B 0.000, C 0.000 }
gfCNCPoint5[23802] = {X 420.6473, Y 16.7687, Z -7.1667, A 0.000, B 0.000, C 0.000 }
gfCNCPoint5[23803] = {X 419.8882, Y 17.7814, Z -7.1667, A 0.000, B 0.000, C 0.000 }
gfCNCPoint5[23804] = {X 419.2035, Y 18.8457, Z -7.1667, A 0.000, B 0.000, C 0.000 }
gfCNCPoint5[23805] = {X 417.7223, Y 21.2434, Z -7.1667, A 0.000, B 0.000, C 0.000 }
gfCNCPoint5[23806] = {X 415.8798, Y 24.2026, Z -7.1667, A 0.000, B 0.000, C 0.000 }
gfCNCPoint5[23807] = {X 419.3433, Y 26.3591, Z -7.1667, A 0.000, B 0.000, C 0.000 }
gfCNCPoint5[23808] = {X 419.3433, Y 26.3591, Z -4.1667, A 0.000, B 0.000, C 0.000 }
gfCNCPoint5[23809] = {X 419.3433, Y 26.3591, Z 11.0000, A 0.000, B 0.000, C 0.000 }
gfCNCPoint5[23810] = {X 352.3575, Y -3.5287, Z 11.0000, A 0.000, B 0.000, C 0.000 }
gfCNCPoint5[23811] = {X 352.3575, Y -3.5287, Z -4.1667, A 0.000, B 0.000, C 0.000 }
gfCNCPoint5[23812] = {X 352.3575, Y -3.5287, Z -7.1667, A 0.000, B 0.000, C 0.000 }
gfCNCPoint5[23813] = {X 351.6041, Y 0.4811, Z -7.1667, A 0.000, B 0.000, C 0.000 }
gfCNCPoint5[23814] = {X 351.8712, Y 0.5313, Z -7.1667, A 0.000, B 0.000, C 0.000 }
gfCNCPoint5[23815] = {X 353.9928, Y 1.0746, Z -7.1667, A 0.000, B 0.000, C 0.000 }
gfCNCPoint5[23816] = {X 356.0464, Y 1.8357, Z -7.1667, A 0.000, B 0.000, C 0.000 }
gfCNCPoint5[23817] = {X 358.0097, Y 2.8062, Z -7.1667, A 0.000, B 0.000, C 0.000 }
gfCNCPoint5[23818] = {X 359.8614, Y 3.9757, Z -7.1667, A 0.000, B 0.000, C 0.000 }
gfCNCPoint5[23819] = {X 361.5814, Y 5.3315, Z -7.1667, A 0.000, B 0.000, C 0.000 }
gfCNCPoint5[23820] = {X 363.1510, Y 6.8589, Z -7.1667, A 0.000, B 0.000, C 0.000 }
gfCNCPoint5[23821] = {X 364.6973, Y 8.7288, Z -7.1667, A 0.000, B 0.000, C 0.000 }
gfCNCPoint5[23822] = {X 366.0539, Y 10.7406, Z -7.1667, A 0.000, B 0.000, C 0.000 }
gfCNCPoint5[23823] = {X 367.2078, Y 12.8751, Z -7.1667, A 0.000, B 0.000, C 0.000 }
gfCNCPoint5[23824] = {X 368.1481, Y 15.1120, Z -7.1667, A 0.000, B 0.000, C 0.000 }
gfCNCPoint5[23825] = {X 368.8658, Y 17.4299, Z -7.1667, A 0.000, B 0.000, C 0.000 }
gfCNCPoint5[23826] = {X 369.3480, Y 19.7226, Z -7.1667, A 0.000, B 0.000, C 0.000 }
gfCNCPoint5[23827] = {X 369.6589, Y 22.0447, Z -7.1667, A 0.000, B 0.000, C 0.000 }
gfCNCPoint5[23828] = {X 369.7968, Y 24.3835, Z -7.1667, A 0.000, B 0.000, C 0.000 }
gfCNCPoint5[23829] = {X 369.7610, Y 26.7261, Z -7.1667, A 0.000, B 0.000, C 0.000 }
gfCNCPoint5[23830] = {X 369.5517, Y 29.0596, Z -7.1667, A 0.000, B 0.000, C 0.000 }
gfCNCPoint5[23831] = {X 369.1700, Y 31.3712, Z -7.1667, A 0.000, B 0.000, C 0.000 }
gfCNCPoint5[23832] = {X 368.6459, Y 33.4754, Z -7.1667, A 0.000, B 0.000, C 0.000 }
gfCNCPoint5[23833] = {X 367.9381, Y 35.5252, Z -7.1667, A 0.000, B 0.000, C 0.000 }
gfCNCPoint5[23834] = {X 367.0520, Y 37.5044, Z -7.1667, A 0.000, B 0.000, C 0.000 }
gfCNCPoint5[23835] = {X 365.9946, Y 39.3977, Z -7.1667, A 0.000, B 0.000, C 0.000 }
gfCNCPoint5[23836] = {X 364.7742, Y 41.1902, Z -7.1667, A 0.000, B 0.000, C 0.000 }
gfCNCPoint5[23837] = {X 364.6579, Y 41.3491, Z -7.1667, A 0.000, B 0.000, C 0.000 }
gfCNCPoint5[23838] = {X 363.2575, Y 43.0261, Z -7.1667, A 0.000, B 0.000, C 0.000 }
gfCNCPoint5[23839] = {X 361.6976, Y 44.5557, Z -7.1667, A 0.000, B 0.000, C 0.000 }
gfCNCPoint5[23840] = {X 359.9935, Y 45.9230, Z -7.1667, A 0.000, B 0.000, C 0.000 }
gfCNCPoint5[23841] = {X 358.1622, Y 47.1144, Z -7.1667, A 0.000, B 0.000, C 0.000 }
gfCNCPoint5[23842] = {X 356.2216, Y 48.1182, Z -7.1667, A 0.000, B 0.000, C 0.000 }
gfCNCPoint5[23843] = {X 354.0239, Y 48.9385, Z -7.1667, A 0.000, B 0.000, C 0.000 }
gfCNCPoint5[23844] = {X 351.7542, Y 49.5309, Z -7.1667, A 0.000, B 0.000, C 0.000 }
gfCNCPoint5[23845] = {X 349.4359, Y 49.8893, Z -7.1667, A 0.000, B 0.000, C 0.000 }
gfCNCPoint5[23846] = {X 347.0933, Y 50.0099, Z -7.1667, A 0.000, B 0.000, C 0.000 }
gfCNCPoint5[23847] = {X 345.0267, Y 49.9751, Z -7.1667, A 0.000, B 0.000, C 0.000 }
gfCNCPoint5[23848] = {X 342.9709, Y 49.7611, Z -7.1667, A 0.000, B 0.000, C 0.000 }
gfCNCPoint5[23849] = {X 340.9414, Y 49.3696, Z -7.1667, A 0.000, B 0.000, C 0.000 }
gfCNCPoint5[23850] = {X 338.9535, Y 48.8036, Z -7.1667, A 0.000, B 0.000, C 0.000 }
gfCNCPoint5[23851] = {X 337.0222, Y 48.0674, Z -7.1667, A 0.000, B 0.000, C 0.000 }
gfCNCPoint5[23852] = {X 335.1620, Y 47.1663, Z -7.1667, A 0.000, B 0.000, C 0.000 }
gfCNCPoint5[23853] = {X 333.5781, Y 46.1881, Z -7.1667, A 0.000, B 0.000, C 0.000 }
gfCNCPoint5[23854] = {X 332.0751, Y 45.0894, Z -7.1667, A 0.000, B 0.000, C 0.000 }
gfCNCPoint5[23855] = {X 330.6624, Y 43.8770, Z -7.1667, A 0.000, B 0.000, C 0.000 }
gfCNCPoint5[23856] = {X 329.7213, Y 43.8764, Z -7.1667, A 0.000, B 0.000, C 0.000 }
gfCNCPoint5[23857] = {X 328.8027, Y 43.6721, Z -7.1667, A 0.000, B 0.000, C 0.000 }
gfCNCPoint5[23858] = {X 327.9501, Y 43.2738, Z -7.1667, A 0.000, B 0.000, C 0.000 }
gfCNCPoint5[23859] = {X 327.2040, Y 42.7002, Z -7.1667, A 0.000, B 0.000, C 0.000 }
gfCNCPoint5[23860] = {X 326.5808, Y 42.0925, Z -7.1667, A 0.000, B 0.000, C 0.000 }
gfCNCPoint5[23861] = {X 325.9523, Y 41.3190, Z -7.1667, A 0.000, B 0.000, C 0.000 }
gfCNCPoint5[23862] = {X 325.5179, Y 40.4220, Z -7.1667, A 0.000, B 0.000, C 0.000 }
gfCNCPoint5[23863] = {X 325.3006, Y 39.4493, Z -7.1667, A 0.000, B 0.000, C 0.000 }
gfCNCPoint5[23864] = {X 325.3120, Y 38.4527, Z -7.1667, A 0.000, B 0.000, C 0.000 }
gfCNCPoint5[23865] = {X 325.5514, Y 37.4852, Z -7.1667, A 0.000, B 0.000, C 0.000 }
gfCNCPoint5[23866] = {X 326.0062, Y 36.5984, Z -7.1667, A 0.000, B 0.000, C 0.000 }
gfCNCPoint5[23867] = {X 330.2396, Y 30.2687, Z -7.1667, A 0.000, B 0.000, C 0.000 }
gfCNCPoint5[23868] = {X 330.8410, Y 29.5517, Z -7.1667, A 0.000, B 0.000, C 0.000 }
gfCNCPoint5[23869] = {X 331.5827, Y 28.9811, Z -7.1667, A 0.000, B 0.000, C 0.000 }
gfCNCPoint5[23870] = {X 332.4299, Y 28.5837, Z -7.1667, A 0.000, B 0.000, C 0.000 }
gfCNCPoint5[23871] = {X 333.3428, Y 28.3779, Z -7.1667, A 0.000, B 0.000, C 0.000 }
gfCNCPoint5[23872] = {X 334.2785, Y 28.3736, Z -7.1667, A 0.000, B 0.000, C 0.000 }
gfCNCPoint5[23873] = {X 335.1933, Y 28.5709, Z -7.1667, A 0.000, B 0.000, C 0.000 }
gfCNCPoint5[23874] = {X 336.0441, Y 28.9606, Z -7.1667, A 0.000, B 0.000, C 0.000 }
gfCNCPoint5[23875] = {X 336.7910, Y 29.5243, Z -7.1667, A 0.000, B 0.000, C 0.000 }
gfCNCPoint5[23876] = {X 337.4284, Y 30.1382, Z -7.1667, A 0.000, B 0.000, C 0.000 }
gfCNCPoint5[23877] = {X 338.0627, Y 30.9279, Z -7.1667, A 0.000, B 0.000, C 0.000 }
gfCNCPoint5[23878] = {X 338.4958, Y 31.8436, Z -7.1667, A 0.000, B 0.000, C 0.000 }
gfCNCPoint5[23879] = {X 338.7036, Y 32.8350, Z -7.1667, A 0.000, B 0.000, C 0.000 }
gfCNCPoint5[23880] = {X 338.6750, Y 33.8475, Z -7.1667, A 0.000, B 0.000, C 0.000 }
gfCNCPoint5[23881] = {X 339.4934, Y 34.5958, Z -7.1667, A 0.000, B 0.000, C 0.000 }
gfCNCPoint5[23882] = {X 340.6301, Y 35.5019, Z -7.1667, A 0.000, B 0.000, C 0.000 }
gfCNCPoint5[23883] = {X 341.8792, Y 36.2453, Z -7.1667, A 0.000, B 0.000, C 0.000 }
gfCNCPoint5[23884] = {X 343.2177, Y 36.8123, Z -7.1667, A 0.000, B 0.000, C 0.000 }
gfCNCPoint5[23885] = {X 344.6208, Y 37.1923, Z -7.1667, A 0.000, B 0.000, C 0.000 }
gfCNCPoint5[23886] = {X 346.0624, Y 37.3785, Z -7.1667, A 0.000, B 0.000, C 0.000 }
gfCNCPoint5[23887] = {X 347.5160, Y 37.3672, Z -7.1667, A 0.000, B 0.000, C 0.000 }
gfCNCPoint5[23888] = {X 348.9570, Y 37.1741, Z -7.1667, A 0.000, B 0.000, C 0.000 }
gfCNCPoint5[23889] = {X 350.3473, Y 36.7489, Z -7.1667, A 0.000, B 0.000, C 0.000 }
gfCNCPoint5[23890] = {X 351.6497, Y 36.1027, Z -7.1667, A 0.000, B 0.000, C 0.000 }
gfCNCPoint5[23891] = {X 352.8295, Y 35.2531, Z -7.1667, A 0.000, B 0.000, C 0.000 }
gfCNCPoint5[23892] = {X 353.9826, Y 34.1325, Z -7.1667, A 0.000, B 0.000, C 0.000 }
gfCNCPoint5[23893] = {X 354.9806, Y 32.8717, Z -7.1667, A 0.000, B 0.000, C 0.000 }
gfCNCPoint5[23894] = {X 355.8065, Y 31.4920, Z -7.1667, A 0.000, B 0.000, C 0.000 }
gfCNCPoint5[23895] = {X 356.4462, Y 30.0168, Z -7.1667, A 0.000, B 0.000, C 0.000 }
gfCNCPoint5[23896] = {X 356.8891, Y 28.4711, Z -7.1667, A 0.000, B 0.000, C 0.000 }
gfCNCPoint5[23897] = {X 357.1624, Y 26.7828, Z -7.1667, A 0.000, B 0.000, C 0.000 }
gfCNCPoint5[23898] = {X 357.2737, Y 25.0763, Z -7.1667, A 0.000, B 0.000, C 0.000 }
gfCNCPoint5[23899] = {X 357.2220, Y 23.3669, Z -7.1667, A 0.000, B 0.000, C 0.000 }
gfCNCPoint5[23900] = {X 357.0079, Y 21.6701, Z -7.1667, A 0.000, B 0.000, C 0.000 }
gfCNCPoint5[23901] = {X 356.6542, Y 20.1543, Z -7.1667, A 0.000, B 0.000, C 0.000 }
gfCNCPoint5[23902] = {X 356.1047, Y 18.6980, Z -7.1667, A 0.000, B 0.000, C 0.000 }
gfCNCPoint5[23903] = {X 355.3688, Y 17.3265, Z -7.1667, A 0.000, B 0.000, C 0.000 }
gfCNCPoint5[23904] = {X 354.4594, Y 16.0633, Z -7.1667, A 0.000, B 0.000, C 0.000 }
gfCNCPoint5[23905] = {X 353.5887, Y 15.1363, Z -7.1667, A 0.000, B 0.000, C 0.000 }
gfCNCPoint5[23906] = {X 352.5980, Y 14.3390, Z -7.1667, A 0.000, B 0.000, C 0.000 }
gfCNCPoint5[23907] = {X 351.5062, Y 13.6868, Z -7.1667, A 0.000, B 0.000, C 0.000 }
gfCNCPoint5[23908] = {X 350.3346, Y 13.1923, Z -7.1667, A 0.000, B 0.000, C 0.000 }
gfCNCPoint5[23909] = {X 349.1057, Y 12.8650, Z -7.1667, A 0.000, B 0.000, C 0.000 }
gfCNCPoint5[23910] = {X 347.3454, Y 12.6451, Z -7.1667, A 0.000, B 0.000, C 0.000 }
gfCNCPoint5[23911] = {X 345.5715, Y 12.6604, Z -7.1667, A 0.000, B 0.000, C 0.000 }
gfCNCPoint5[23912] = {X 343.8153, Y 12.9104, Z -7.1667, A 0.000, B 0.000, C 0.000 }
gfCNCPoint5[23913] = {X 342.1076, Y 13.3910, Z -7.1667, A 0.000, B 0.000, C 0.000 }
gfCNCPoint5[23914] = {X 340.4787, Y 14.0935, Z -7.1667, A 0.000, B 0.000, C 0.000 }
gfCNCPoint5[23915] = {X 338.9572, Y 15.0056, Z -7.1667, A 0.000, B 0.000, C 0.000 }
gfCNCPoint5[23916] = {X 338.9182, Y 15.8503, Z -7.1667, A 0.000, B 0.000, C 0.000 }
gfCNCPoint5[23917] = {X 338.7154, Y 16.6712, Z -7.1667, A 0.000, B 0.000, C 0.000 }
gfCNCPoint5[23918] = {X 338.3565, Y 17.4369, Z -7.1667, A 0.000, B 0.000, C 0.000 }
gfCNCPoint5[23919] = {X 337.8554, Y 18.1180, Z -7.1667, A 0.000, B 0.000, C 0.000 }
gfCNCPoint5[23920] = {X 337.2312, Y 18.6885, Z -7.1667, A 0.000, B 0.000, C 0.000 }
gfCNCPoint5[23921] = {X 336.5140, Y 19.2162, Z -7.1667, A 0.000, B 0.000, C 0.000 }
gfCNCPoint5[23922] = {X 335.6982, Y 19.6754, Z -7.1667, A 0.000, B 0.000, C 0.000 }
gfCNCPoint5[23923] = {X 334.8027, Y 19.9480, Z -7.1667, A 0.000, B 0.000, C 0.000 }
gfCNCPoint5[23924] = {X 333.8694, Y 20.0213, Z -7.1667, A 0.000, B 0.000, C 0.000 }
gfCNCPoint5[23925] = {X 332.9422, Y 19.8919, Z -7.1667, A 0.000, B 0.000, C 0.000 }
gfCNCPoint5[23926] = {X 332.0647, Y 19.5657, Z -7.1667, A 0.000, B 0.000, C 0.000 }
gfCNCPoint5[23927] = {X 331.2781, Y 19.0581, Z -7.1667, A 0.000, B 0.000, C 0.000 }
gfCNCPoint5[23928] = {X 330.6193, Y 18.3931, Z -7.1667, A 0.000, B 0.000, C 0.000 }
gfCNCPoint5[23929] = {X 330.1192, Y 17.6017, Z -7.1667, A 0.000, B 0.000, C 0.000 }
gfCNCPoint5[23930] = {X 326.5942, Y 10.3502, Z -7.1667, A 0.000, B 0.000, C 0.000 }
gfCNCPoint5[23931] = {X 326.2930, Y 9.5271, Z -7.1667, A 0.000, B 0.000, C 0.000 }
gfCNCPoint5[23932] = {X 326.1640, Y 8.6602, Z -7.1667, A 0.000, B 0.000, C 0.000 }
gfCNCPoint5[23933] = {X 326.2128, Y 7.7851, Z -7.1667, A 0.000, B 0.000, C 0.000 }
gfCNCPoint5[23934] = {X 326.4371, Y 6.9378, Z -7.1667, A 0.000, B 0.000, C 0.000 }
gfCNCPoint5[23935] = {X 326.8279, Y 6.1532, Z -7.1667, A 0.000, B 0.000, C 0.000 }
gfCNCPoint5[23936] = {X 327.3690, Y 5.4637, Z -7.1667, A 0.000, B 0.000, C 0.000 }
gfCNCPoint5[23937] = {X 328.0381, Y 4.8976, Z -7.1667, A 0.000, B 0.000, C 0.000 }
gfCNCPoint5[23938] = {X 328.7084, Y 4.4386, Z -7.1667, A 0.000, B 0.000, C 0.000 }
gfCNCPoint5[23939] = {X 329.5887, Y 3.9824, Z -7.1667, A 0.000, B 0.000, C 0.000 }
gfCNCPoint5[23940] = {X 330.5498, Y 3.7389, Z -7.1667, A 0.000, B 0.000, C 0.000 }
gfCNCPoint5[23941] = {X 331.5411, Y 3.7209, Z -7.1667, A 0.000, B 0.000, C 0.000 }
gfCNCPoint5[23942] = {X 332.5104, Y 3.9295, Z -7.1667, A 0.000, B 0.000, C 0.000 }
gfCNCPoint5[23943] = {X 334.1674, Y 3.0112, Z -7.1667, A 0.000, B 0.000, C 0.000 }
gfCNCPoint5[23944] = {X 335.8816, Y 2.2048, Z -7.1667, A 0.000, B 0.000, C 0.000 }
gfCNCPoint5[23945] = {X 337.9832, Y 1.3861, Z -7.1667, A 0.000, B 0.000, C 0.000 }
gfCNCPoint5[23946] = {X 340.1471, Y 0.7505, Z -7.1667, A 0.000, B 0.000, C 0.000 }
gfCNCPoint5[23947] = {X 342.3576, Y 0.3024, Z -7.1667, A 0.000, B 0.000, C 0.000 }
gfCNCPoint5[23948] = {X 344.5983, Y 0.0452, Z -7.1667, A 0.000, B 0.000, C 0.000 }
gfCNCPoint5[23949] = {X 346.8528, Y -0.0191, Z -7.1667, A 0.000, B 0.000, C 0.000 }
gfCNCPoint5[23950] = {X 349.1045, Y 0.1097, Z -7.1667, A 0.000, B 0.000, C 0.000 }
gfCNCPoint5[23951] = {X 351.3369, Y 0.4309, Z -7.1667, A 0.000, B 0.000, C 0.000 }
gfCNCPoint5[23952] = {X 351.6041, Y 0.4811, Z -7.1667, A 0.000, B 0.000, C 0.000 }
gfCNCPoint5[23953] = {X 352.3427, Y -3.4501, Z -7.1667, A 0.000, B 0.000, C 0.000 }
gfCNCPoint5[23954] = {X 351.5893, Y 0.5597, Z -7.1667, A 0.000, B 0.000, C 0.000 }
gfCNCPoint5[23955] = {X 351.8559, Y 0.6098, Z -7.1667, A 0.000, B 0.000, C 0.000 }
gfCNCPoint5[23956] = {X 353.9694, Y 1.1511, Z -7.1667, A 0.000, B 0.000, C 0.000 }
gfCNCPoint5[23957] = {X 356.0151, Y 1.9093, Z -7.1667, A 0.000, B 0.000, C 0.000 }
gfCNCPoint5[23958] = {X 357.9708, Y 2.8761, Z -7.1667, A 0.000, B 0.000, C 0.000 }
gfCNCPoint5[23959] = {X 359.8154, Y 4.0412, Z -7.1667, A 0.000, B 0.000, C 0.000 }
gfCNCPoint5[23960] = {X 361.5287, Y 5.3918, Z -7.1667, A 0.000, B 0.000, C 0.000 }
gfCNCPoint5[23961] = {X 363.0923, Y 6.9132, Z -7.1667, A 0.000, B 0.000, C 0.000 }
gfCNCPoint5[23962] = {X 364.6335, Y 8.7771, Z -7.1667, A 0.000, B 0.000, C 0.000 }
gfCNCPoint5[23963] = {X 365.9856, Y 10.7824, Z -7.1667, A 0.000, B 0.000, C 0.000 }
gfCNCPoint5[23964] = {X 367.1358, Y 12.9099, Z -7.1667, A 0.000, B 0.000, C 0.000 }
gfCNCPoint5[23965] = {X 368.0730, Y 15.1395, Z -7.1667, A 0.000, B 0.000, C 0.000 }
gfCNCPoint5[23966] = {X 368.7884, Y 17.4498, Z -7.1667, A 0.000, B 0.000, C 0.000 }
gfCNCPoint5[23967] = {X 369.2692, Y 19.7366, Z -7.1667, A 0.000, B 0.000, C 0.000 }
gfCNCPoint5[23968] = {X 369.5793, Y 22.0528, Z -7.1667, A 0.000, B 0.000, C 0.000 }
gfCNCPoint5[23969] = {X 369.7168, Y 24.3856, Z -7.1667, A 0.000, B 0.000, C 0.000 }
gfCNCPoint5[23970] = {X 369.6811, Y 26.7222, Z -7.1667, A 0.000, B 0.000, C 0.000 }
gfCNCPoint5[23971] = {X 369.4723, Y 29.0496, Z -7.1667, A 0.000, B 0.000, C 0.000 }
gfCNCPoint5[23972] = {X 369.0916, Y 31.3553, Z -7.1667, A 0.000, B 0.000, C 0.000 }
gfCNCPoint5[23973] = {X 368.5692, Y 33.4527, Z -7.1667, A 0.000, B 0.000, C 0.000 }
gfCNCPoint5[23974] = {X 367.8636, Y 35.4959, Z -7.1667, A 0.000, B 0.000, C 0.000 }
gfCNCPoint5[23975] = {X 366.9804, Y 37.4687, Z -7.1667, A 0.000, B 0.000, C 0.000 }
gfCNCPoint5[23976] = {X 365.9264, Y 39.3559, Z -7.1667, A 0.000, B 0.000, C 0.000 }
gfCNCPoint5[23977] = {X 364.7099, Y 41.1426, Z -7.1667, A 0.000, B 0.000, C 0.000 }
gfCNCPoint5[23978] = {X 364.5937, Y 41.3014, Z -7.1667, A 0.000, B 0.000, C 0.000 }
gfCNCPoint5[23979] = {X 363.1985, Y 42.9720, Z -7.1667, A 0.000, B 0.000, C 0.000 }
gfCNCPoint5[23980] = {X 361.6445, Y 44.4959, Z -7.1667, A 0.000, B 0.000, C 0.000 }
gfCNCPoint5[23981] = {X 359.9468, Y 45.8581, Z -7.1667, A 0.000, B 0.000, C 0.000 }
gfCNCPoint5[23982] = {X 358.1224, Y 47.0450, Z -7.1667, A 0.000, B 0.000, C 0.000 }
gfCNCPoint5[23983] = {X 356.1891, Y 48.0451, Z -7.1667, A 0.000, B 0.000, C 0.000 }
gfCNCPoint5[23984] = {X 353.9990, Y 48.8624, Z -7.1667, A 0.000, B 0.000, C 0.000 }
gfCNCPoint5[23985] = {X 351.7371, Y 49.4527, Z -7.1667, A 0.000, B 0.000, C 0.000 }
gfCNCPoint5[23986] = {X 349.4268, Y 49.8098, Z -7.1667, A 0.000, B 0.000, C 0.000 }
gfCNCPoint5[23987] = {X 347.0922, Y 49.9299, Z -7.1667, A 0.000, B 0.000, C 0.000 }
gfCNCPoint5[23988] = {X 345.0325, Y 49.8953, Z -7.1667, A 0.000, B 0.000, C 0.000 }
gfCNCPoint5[23989] = {X 342.9835, Y 49.6821, Z -7.1667, A 0.000, B 0.000, C 0.000 }
gfCNCPoint5[23990] = {X 340.9608, Y 49.2920, Z -7.1667, A 0.000, B 0.000, C 0.000 }
gfCNCPoint5[23991] = {X 338.9796, Y 48.7280, Z -7.1667, A 0.000, B 0.000, C 0.000 }
gfCNCPoint5[23992] = {X 337.0547, Y 47.9942, Z -7.1667, A 0.000, B 0.000, C 0.000 }
gfCNCPoint5[23993] = {X 335.2007, Y 47.0963, Z -7.1667, A 0.000, B 0.000, C 0.000 }
gfCNCPoint5[23994] = {X 333.6121, Y 46.1146, Z -7.1667, A 0.000, B 0.000, C 0.000 }
